(* IEC 61131-3 sources: Industry-PLC-LLM/data/PLCBEAD_repo/PLCBEAD_PLCEmbed-main/PLC-BEAD/Source/OpenPLCv2 (part 8) *)

(* ---- REPLACE_CHARS.ST ---- *)
FUNCTION_BLOCK REPLACE_CHARS_Block

	VAR_INPUT
		STR :	STRING;
		SRC :	STRING;
		REP :	STRING;
	END_VAR

	VAR_OUTPUT
		REPLACE_CHARS :	STRING;
	END_VAR

	VAR
		tmp :	STRING;
		a :	INT;
		b :	INT;
		c :	STRING;
		stp :	INT;
	END_VAR

	REPLACE_CHARS := STR;

	a := LEN(src);
	b := LEN(rep);
	IF a < b THEN
		rep := LEFT(rep, a);
	ELSIF b < a THEN
		src := LEFT(src, b);
	END_IF;

	stp := LEN(str);
	FOR a := 1 TO stp DO
		c := MID(REPLACE_CHARS, 1, a);
		b := FIND(src, c);
		IF b > 0 THEN
			tmp := MID(rep, 1, b);
			REPLACE_CHARS := REPLACE(REPLACE_CHARS, tmp, 1, a);
		END_IF;
	END_FOR;

END_FUNCTION_BLOCK

PROGRAM program0

	VAR
		STR :	STRING;
		SRC :	STRING;
		REP :	STRING;

        REPLACE_CHARS :	STRING;
		func_block : REPLACE_CHARS_Block;
	END_VAR
		func_block.STR := STR;
		func_block.SRC := SRC;
		func_block.REP := REP;
		func_block();
		REPLACE_CHARS := func_block.REPLACE_CHARS;

END_PROGRAM

CONFIGURATION Config0

	RESOURCE Res0 ON PLC
		TASK task0(INTERVAL := T#20ms,PRIORITY := 0);
		PROGRAM instance0 WITH task0 : program0;
	END_RESOURCE

END_CONFIGURATION

(* ---- RMP_B.ST ---- *)
FUNCTION TIME_TO_UDINT2:UDINT
	VAR_INPUT
		X :	TIME;
	END_VAR

	TIME_TO_UDINT2 := DINT_TO_UDINT(TIME_TO_DINT(X));
END_FUNCTION

FUNCTION_BLOCK T_PLC_MS_block
	VAR_OUTPUT
		T_PLC_MS :	UDINT;
	END_VAR

	VAR_EXTERNAL
		PLC_TICKS_PER_SEC :	INT;
		PLC_SYS_TICK_CNT :	DINT;
	END_VAR

	VAR
		debug :	BOOL;(*Debug-Mode ON / OFF*)
		N :	INT;(*Debug-Faktor*)
		Offset :	UDINT;(*Debug-Offset*)
		temp :	DWORD := DWORD#1;(*Debug-Offset*)
		mode :	BOOL;(*modus*)
		faktor :	UDINT;(*Systemtakt-Faktor*)
		init :	BOOL;
		v_plc_ticks_per_sec :	UDINT;
		base :	UDINT := UDINT#1000;
	END_VAR

	IF init = FALSE THEN
		v_plc_ticks_per_sec := INT_TO_UDINT(PLC_TICKS_PER_SEC);
		IF v_plc_ticks_per_sec = UDINT#1024 THEN
			faktor := UDINT#1;
			mode := FALSE;
		ELSIF v_plc_ticks_per_sec > UDINT#0 THEN
			IF v_plc_ticks_per_sec <= base THEN
				faktor := base / v_plc_ticks_per_sec;
				mode := FALSE;
			ELSE
				faktor := v_plc_ticks_per_sec / base;
				mode := TRUE;
			END_IF;
		ELSE
			faktor := UDINT#1;
		END_IF;
		init := TRUE;
	END_IF;

	IF mode THEN
		T_PLC_MS := DINT_TO_UDINT(PLC_SYS_TICK_CNT) / faktor;
	ELSE
		T_PLC_MS := DINT_TO_UDINT(PLC_SYS_TICK_CNT) * faktor;
	END_IF;

	IF debug THEN
		T_PLC_MS := (DWORD_TO_UDINT(SHL(UDINT_TO_DWORD(T_PLC_MS),N) OR SHL(temp,N)) - UDINT#1) + Offset;
	END_IF;
END_FUNCTION_BLOCK

FUNCTION FRMP_B:BYTE
	VAR_INPUT
		START :	BYTE;
		DIR :	BOOL;
		TD :	TIME;
		TR :	TIME;
	END_VAR

	IF TD < TR THEN
		FRMP_B := MIN(UDINT_TO_BYTE(DWORD_TO_UDINT(SHL(TIME_TO_DWORD(TD), 8)) / TIME_TO_UDINT2(TR)), SEL(DIR, START, USINT_TO_BYTE(USINT#255 - BYTE_TO_USINT(START))));
		IF DIR THEN
			FRMP_B := USINT_TO_BYTE(BYTE_TO_USINT(START) + BYTE_TO_USINT(FRMP_B));
		ELSE
			FRMP_B := USINT_TO_BYTE(BYTE_TO_USINT(START) - BYTE_TO_USINT(FRMP_B));
		END_IF;
	ELSE
		FRMP_B := SEL(DIR, BYTE#0, BYTE#255);
	END_IF;
END_FUNCTION

FUNCTION_BLOCK _RMP_B
	VAR_INPUT
		DIR :	BOOL;
		E :	BOOL := TRUE;
		TR :	TIME;
	END_VAR

	VAR_IN_OUT
		RMP :	BYTE;
	END_VAR

	VAR
		T_PLC_MS :	T_PLC_MS_block;
		tx :	TIME;
		tl :	TIME;
		tn :	TIME;
		init :	BOOL;
		last_dir :	BOOL;
		start :	BYTE;
	END_VAR

	T_PLC_MS();
	tx := UDINT_TO_TIME(T_PLC_MS.T_PLC_MS);

	IF E AND init AND (dir = last_dir) AND (RMP <> SEL(DIR, BYTE#0, BYTE#255)) AND TR = tn THEN
		RMP := FRMP_B(start, DIR, tx - tl, TR);
	ELSE
		init := TRUE;
		tl := tx;
		tn := tr;
		start := RMP;
	END_IF;
	last_dir := dir;
END_FUNCTION_BLOCK

FUNCTION_BLOCK RMP_B_Block

	VAR_INPUT
		SET :	BOOL;
		PT :	TIME;
		E :	BOOL := TRUE;
		UP :	BOOL := TRUE;
		RST :	BOOL;
	END_VAR

	VAR_OUTPUT
		OUT :	BYTE;
		BUSY :	BOOL;
		HIGH :	BOOL;
		LOW :	BOOL;
	END_VAR

	VAR
		rmp :	_RMP_B;
	END_VAR

	rmp(dir := UP, E := E, TR := PT, RMP := out);
	out := rmp.RMP;

	IF RST THEN
		out := BYTE#0;
	ELSIF SET THEN
		out := BYTE#255;
	END_IF;

low := out = BYTE#0;
high := out = BYTE#255;
busy := NOT (low OR high) AND E;

END_FUNCTION_BLOCK

PROGRAM program0
	VAR
		SET :	BOOL;
		PT :	TIME;
		E :	BOOL := TRUE;
		UP :	BOOL := TRUE;
		RST :	BOOL;

		OUT :	BYTE;
		BUSY :	BOOL;
		HIGH :	BOOL;
		LOW :	BOOL;

		func_block : RMP_B_Block;
	END_VAR
		func_block.SET := SET;
		func_block.PT := PT;
		func_block.E := E;
		func_block.UP := UP;
		func_block.RST := RST;
		func_block();
		OUT := func_block.OUT;
		BUSY := func_block.BUSY;
		HIGH := func_block.HIGH;
		LOW := func_block.LOW;

END_PROGRAM

CONFIGURATION Config0
	VAR_GLOBAL
		PLC_TICKS_PER_SEC :	INT;
		PLC_SYS_TICK_CNT :	DINT;
	END_VAR

  	RESOURCE Res0 ON PLC
    	TASK task0(INTERVAL := T#20ms,PRIORITY := 0);
    	PROGRAM instance0 WITH task0 : program0;
  	END_RESOURCE
END_CONFIGURATION

(* ---- RMP_SOFT.ST ---- *)
FUNCTION TIME_TO_UDINT2:UDINT
	VAR_INPUT
		X :	TIME;
	END_VAR

	TIME_TO_UDINT2 := DINT_TO_UDINT(TIME_TO_DINT(X));
END_FUNCTION

FUNCTION_BLOCK T_PLC_MS_block
	VAR_OUTPUT
		T_PLC_MS :	UDINT;
	END_VAR

	VAR_EXTERNAL
		PLC_TICKS_PER_SEC :	INT;
		PLC_SYS_TICK_CNT :	DINT;
	END_VAR

	VAR
		debug :	BOOL;(*Debug-Mode ON / OFF*)
		N :	INT;(*Debug-Faktor*)
		Offset :	UDINT;(*Debug-Offset*)
		temp :	DWORD := DWORD#1;(*Debug-Offset*)
		mode :	BOOL;(*modus*)
		faktor :	UDINT;(*Systemtakt-Faktor*)
		init :	BOOL;
		v_plc_ticks_per_sec :	UDINT;
		base :	UDINT := UDINT#1000;
	END_VAR

	IF init = FALSE THEN
		v_plc_ticks_per_sec := INT_TO_UDINT(PLC_TICKS_PER_SEC);
		IF v_plc_ticks_per_sec = UDINT#1024 THEN
			faktor := UDINT#1;
			mode := FALSE;
		ELSIF v_plc_ticks_per_sec > UDINT#0 THEN
			IF v_plc_ticks_per_sec <= base THEN
				faktor := base / v_plc_ticks_per_sec;
				mode := FALSE;
			ELSE
				faktor := v_plc_ticks_per_sec / base;
				mode := TRUE;
			END_IF;
		ELSE
			faktor := UDINT#1;
		END_IF;
		init := TRUE;
	END_IF;

	IF mode THEN
		T_PLC_MS := DINT_TO_UDINT(PLC_SYS_TICK_CNT) / faktor;
	ELSE
		T_PLC_MS := DINT_TO_UDINT(PLC_SYS_TICK_CNT) * faktor;
	END_IF;

	IF debug THEN
		T_PLC_MS := (DWORD_TO_UDINT(SHL(UDINT_TO_DWORD(T_PLC_MS),N) OR SHL(temp,N)) - UDINT#1) + Offset;
	END_IF;
END_FUNCTION_BLOCK

FUNCTION FRMP_B:BYTE
	VAR_INPUT
		START :	BYTE;
		DIR :	BOOL;
		TD :	TIME;
		TR :	TIME;
	END_VAR

	IF TD < TR THEN
		FRMP_B := MIN(UDINT_TO_BYTE(DWORD_TO_UDINT(SHL(TIME_TO_DWORD(TD), 8)) / TIME_TO_UDINT2(TR)), SEL(DIR, START, USINT_TO_BYTE(USINT#255 - BYTE_TO_USINT(START))));
		IF DIR THEN
			FRMP_B := USINT_TO_BYTE(BYTE_TO_USINT(START) + BYTE_TO_USINT(FRMP_B));
		ELSE
			FRMP_B := USINT_TO_BYTE(BYTE_TO_USINT(START) - BYTE_TO_USINT(FRMP_B));
		END_IF;
	ELSE
		FRMP_B := SEL(DIR, BYTE#0, BYTE#255);
	END_IF;
END_FUNCTION

FUNCTION_BLOCK _RMP_B
	VAR_INPUT
		DIR :	BOOL;
		E :	BOOL := TRUE;
		TR :	TIME;
	END_VAR

	VAR_IN_OUT
		RMP :	BYTE;
	END_VAR

	VAR
		T_PLC_MS :	T_PLC_MS_block;
		tx :	TIME;
		tl :	TIME;
		tn :	TIME;
		init :	BOOL;
		last_dir :	BOOL;
		start :	BYTE;
	END_VAR

	T_PLC_MS();
	tx := UDINT_TO_TIME(T_PLC_MS.T_PLC_MS);

	IF E AND init AND (dir = last_dir) AND (RMP <> SEL(DIR, BYTE#0, BYTE#255)) AND TR = tn THEN
		RMP := FRMP_B(start, DIR, tx - tl, TR);
	ELSE
		init := TRUE;
		tl := tx;
		tn := tr;
		start := RMP;
	END_IF;
	last_dir := dir;
END_FUNCTION_BLOCK

FUNCTION_BLOCK RMP_SOFT_Block

	VAR_INPUT
		IN :	BOOL;
		VAL :	BYTE;
		PT_ON :	TIME := T#100ms;
		PT_OFF :	TIME := T#100ms;
	END_VAR

	VAR_OUTPUT
		OUT :	BYTE := BYTE#00;
	END_VAR

	VAR
		rmp :	_RMP_B;
		tmp :	BYTE;
	END_VAR

	tmp := SEL(in, BYTE#0, val);
	IF tmp > out THEN
		(* we need to ramp down *)
		rmp(dir := TRUE, E := TRUE, TR := PT_ON, RMP := out);
		out := rmp.RMP;
		(* make sure out does not surpass tmp *)
		out := MIN(out, tmp);
	ELSIF tmp < out THEN
		(* we need to ramp up *)
		rmp(dir := FALSE, E := TRUE, TR := PT_OFF, RMP := out);
		out := rmp.RMP;
		(* make sure out does not surpass tmp *)
		out := MAX(out, tmp);
	ELSE
		(* no ramp necessary *)
		rmp(E := FALSE, RMP := out);
		out := rmp.RMP;
	END_IF;

END_FUNCTION_BLOCK

PROGRAM program0
	VAR
		IN :	BOOL;
		VAL :	BYTE;
		PT_ON :	TIME;
		PT_OFF : TIME;

		OUT  :	BYTE;

		func_block : RMP_SOFT_Block;
	END_VAR
		func_block.IN := IN;
		func_block.VAL := VAL;
		func_block.PT_ON := PT_ON;
		func_block.PT_OFF := PT_OFF;
		func_block();
		OUT  := func_block.OUT ;

END_PROGRAM

CONFIGURATION Config0
	VAR_GLOBAL
		PLC_TICKS_PER_SEC :	INT;
		PLC_SYS_TICK_CNT :	DINT;
	END_VAR

  	RESOURCE Res0 ON PLC
    	TASK task0(INTERVAL := T#20ms,PRIORITY := 0);
    	PROGRAM instance0 WITH task0 : program0;
  	END_RESOURCE
END_CONFIGURATION

(* ---- RMP_W.ST ---- *)
FUNCTION_BLOCK T_PLC_MS_block
	VAR_OUTPUT
		T_PLC_MS :	UDINT;
	END_VAR

	VAR_EXTERNAL
		PLC_TICKS_PER_SEC :	INT;
		PLC_SYS_TICK_CNT :	DINT;
	END_VAR

	VAR
		debug :	BOOL;(*Debug-Mode ON / OFF*)
		N :	INT;(*Debug-Faktor*)
		Offset :	UDINT;(*Debug-Offset*)
		temp :	DWORD := DWORD#1;(*Debug-Offset*)
		mode :	BOOL;(*modus*)
		faktor :	UDINT;(*Systemtakt-Faktor*)
		init :	BOOL;
		v_plc_ticks_per_sec :	UDINT;
		base :	UDINT := UDINT#1000;
	END_VAR

	IF init = FALSE THEN
		v_plc_ticks_per_sec := INT_TO_UDINT(PLC_TICKS_PER_SEC);
		IF v_plc_ticks_per_sec = UDINT#1024 THEN
			faktor := UDINT#1;
			mode := FALSE;
		ELSIF v_plc_ticks_per_sec > UDINT#0 THEN
			IF v_plc_ticks_per_sec <= base THEN
				faktor := base / v_plc_ticks_per_sec;
				mode := FALSE;
			ELSE
				faktor := v_plc_ticks_per_sec / base;
				mode := TRUE;
			END_IF;
		ELSE
			faktor := UDINT#1;
		END_IF;
		init := TRUE;
	END_IF;

	IF mode THEN
		T_PLC_MS := DINT_TO_UDINT(PLC_SYS_TICK_CNT) / faktor;
	ELSE
		T_PLC_MS := DINT_TO_UDINT(PLC_SYS_TICK_CNT) * faktor;
	END_IF;

	IF debug THEN
		T_PLC_MS := (DWORD_TO_UDINT(SHL(UDINT_TO_DWORD(T_PLC_MS),N) OR SHL(temp,N)) - UDINT#1) + Offset;
	END_IF;
END_FUNCTION_BLOCK

FUNCTION _WORD_TO_DINT:DINT
	VAR_INPUT
		IN :	WORD;
	END_VAR
	_WORD_TO_DINT := UINT_TO_DINT(WORD_TO_UINT(IN));
END_FUNCTION

FUNCTION TIME_TO_UDINT2:UDINT
	VAR_INPUT
		X :	TIME;
	END_VAR

	TIME_TO_UDINT2 := DINT_TO_UDINT(TIME_TO_DINT(X));
END_FUNCTION

FUNCTION_BLOCK _RMP_W

	VAR_INPUT
		DIR :	BOOL;
		E :	BOOL := TRUE;
		TR :	TIME;
	END_VAR

	VAR_IN_OUT
		RMP :	WORD;
	END_VAR

	VAR
		T_PLC_MS :	T_PLC_MS_block;
		tx :	UDINT;
		tl :	UDINT;
		ptesss :	DINT;
		init :	BOOL;
		last_dir :	BOOL;
	END_VAR

	T_PLC_MS();
	tx := T_PLC_MS.T_PLC_MS;
	IF E AND init THEN
		(* we need to set tl = tx when direction changes *)
		IF dir XOR last_dir THEN
			tl := tx;
			last_dir := dir;
		END_IF;
		(* check_elapsed time and calculate only if necessary *)
		IF tr > t#0s THEN
			ptesss := DWORD_TO_DINT(UDINT_TO_DWORD(DWORD_TO_UDINT(SHL(UDINT_TO_DWORD(tx-tl), 16)) / TIME_TO_UDINT2(TR)));
		ELSE
			ptesss := DINT#65535;
		END_IF;
		IF ptesss > DINT#0 THEN
			(* perform the ptesss on the ramp *)
			tl := tx;
			(* calculate the ptesss response *)
			IF NOT dir THEN ptesss := - ptesss; END_IF;
			rmp := DINT_TO_WORD(LIMIT(DINT#0, _WORD_TO_DINT(rmp) + ptesss, DINT#65535));
		END_IF;
	ELSE
		tl := tx;
		init := TRUE;
	END_IF;
END_FUNCTION_BLOCK

FUNCTION_BLOCK RMP_W

	VAR_INPUT
		SET :	BOOL;
		PT :	TIME;
		E :	BOOL := TRUE;
		UP :	BOOL := TRUE;
		RST :	BOOL;
	END_VAR

	VAR_OUTPUT
		OUT :	WORD;
		BUSY :	BOOL;
		HIGH :	BOOL;
		LOW :	BOOL;
	END_VAR

	VAR
		rmp :	_RMP_W;
	END_VAR

	rmp(dir := UP, E := E, TR := PT, rmp := out);
	out := rmp.RMP;

	IF RST THEN
		out := WORD#0;
	ELSIF SET THEN
		out := WORD#65535;
	END_IF;

	low := out = WORD#0;
	high := out = WORD#65535;
	busy := NOT (low OR high) AND E;

END_FUNCTION_BLOCK

PROGRAM program0
  VAR
		SET :	BOOL;
		PT  :	TIME;
		E   :	BOOL;
		UP  :	BOOL ;
		RST :	BOOL;

		OUT  :	WORD;
		BUSY :	BOOL;
		HIGH :	BOOL;
		LOW  :	BOOL;

	func_block : RMP_W;
  END_VAR
	func_block.SET:=SET;
	func_block.PT :=PT ;
	func_block.E  :=E ;
	func_block.UP :=UP ;
	func_block.RST:=RST;
	func_block();
	OUT  := func_block.OUT ;
	BUSY := func_block.BUSY;
	HIGH := func_block.HIGH;
	LOW  := func_block.LOW ;

END_PROGRAM

CONFIGURATION Config0
	VAR_GLOBAL
		PLC_TICKS_PER_SEC :	INT;
		PLC_SYS_TICK_CNT :	DINT;
	END_VAR
  	RESOURCE Res0 ON PLC
    	TASK task0(INTERVAL := T#20ms,PRIORITY := 0);
    	PROGRAM instance0 WITH task0 : program0;
  	END_RESOURCE
END_CONFIGURATION

(* ---- RTC_2.ST ---- *)
FUNCTION _INT_TO_UDINT:UDINT
	VAR_INPUT
		IN :	INT;
	END_VAR

	_INT_TO_UDINT := DINT_TO_UDINT(INT_TO_DINT(IN));
END_FUNCTION

FUNCTION SET_DATE:UDINT

	VAR_INPUT
		YEAR :	INT;
		MONTH :	INT;
		DAY :	INT;
	END_VAR

	VAR
		count :	INT;
	END_VAR

	IF month > 2 THEN
		count := (month - 1) * 30;
		IF month > 7 THEN
			count := count + DWORD_TO_INT(SHR(DINT_TO_DWORD(INT_TO_DINT(month) - INT_TO_DINT(3)),1));
		ELSE
			count := count + DWORD_TO_INT(SHR(DINT_TO_DWORD(INT_TO_DINT(month) - INT_TO_DINT(4)),1));
		END_IF;
		IF SHL(INT_TO_WORD(year),14) = WORD#0 THEN
			count := count + 1;
		END_IF;
	ELSE
		count := (month - 1) * 31;
	END_IF;
	SET_DATE := (_INT_TO_UDINT(count + day - 1) + DWORD_TO_UDINT(SHR(UDINT_TO_DWORD(_INT_TO_UDINT(year) * UDINT#1461 - UDINT#2878169), 2))) * UDINT#86400;

END_FUNCTION

FUNCTION SET_DT:UDINT
	VAR_INPUT
		YEAR :	INT;
		MONTH :	INT;
		DAY :	INT;
		HOUR :	INT;
		MINUTE :	INT;
		SECOND :	INT;
	END_VAR

	SET_DT := SET_DATE(YEAR, MONTH, DAY) + _INT_TO_UDINT(SECOND) + _INT_TO_UDINT(MINUTE) * UDINT#60 + _INT_TO_UDINT(HOUR) * UDINT#3600;
END_FUNCTION

FUNCTION DT_TO_DATE2:UDINT

	VAR_INPUT
		IN :	UDINT;
	END_VAR

	DT_TO_DATE2 := (IN / UDINT#86400) * UDINT#86400;

END_FUNCTION

FUNCTION YEAR_OF_DATE:INT
	VAR_INPUT
		IDATE :	UDINT;
	END_VAR

	YEAR_OF_DATE := UDINT_TO_INT((idate+UDINT#43200) / UDINT#31557600 + UDINT#1970);
END_FUNCTION

FUNCTION DST:BOOL
	VAR_INPUT
		UTC :	UDINT;
	END_VAR

	VAR
		yr :	INT;
		yr4 :	UDINT;
		ltc :	UDINT;
		idate :	UDINT;
	END_VAR

	yr := YEAR_OF_DATE(DT_TO_DATE2(UTC));
	ltc := UTC;
	idate := SET_DT(yr, 3, 31, 1, 0, 0);
	yr4 := DWORD_TO_UDINT(SHR(INT_TO_DWORD(5 * yr), 2)) + UDINT#1;
	DST := (idate - ((yr4 + UDINT#3) MOD UDINT#7) * UDINT#86400 <= ltc) AND (idate + (UDINT#214 - (yr4) MOD UDINT#7) * UDINT#86400 > ltc);

END_FUNCTION

FUNCTION_BLOCK T_PLC_MS_Block
	VAR_OUTPUT
		T_PLC_MS :	UDINT;
	END_VAR

	VAR_EXTERNAL
		PLC_TICKS_PER_SEC :	INT;
		PLC_SYS_TICK_CNT :	DINT;
	END_VAR

	VAR
		debug :	BOOL;(*Debug-Mode ON / OFF*)
		N :	INT;(*Debug-Faktor*)
		Offset :	UDINT;(*Debug-Offset*)
		temp :	DWORD := DWORD#1;(*Debug-Offset*)
		mode :	BOOL;(*modus*)
		faktor :	UDINT;(*Systemtakt-Faktor*)
		init :	BOOL;
		v_plc_ticks_per_sec :	UDINT;
		base :	UDINT := UDINT#1000;
	END_VAR

	IF init = FALSE THEN
		v_plc_ticks_per_sec := INT_TO_UDINT(PLC_TICKS_PER_SEC);
		IF v_plc_ticks_per_sec = UDINT#1024 THEN
			faktor := UDINT#1;
			mode := FALSE;
		ELSIF v_plc_ticks_per_sec > UDINT#0 THEN
			IF v_plc_ticks_per_sec <= base THEN
				faktor := base / v_plc_ticks_per_sec;
				mode := FALSE;
			ELSE
				faktor := v_plc_ticks_per_sec / base;
				mode := TRUE;
			END_IF;
		ELSE
			faktor := UDINT#1;
		END_IF;
		init := TRUE;
	END_IF;

	IF mode THEN
		T_PLC_MS := DINT_TO_UDINT(PLC_SYS_TICK_CNT) / faktor;
	ELSE
		T_PLC_MS := DINT_TO_UDINT(PLC_SYS_TICK_CNT) * faktor;
	END_IF;

	IF debug THEN
		T_PLC_MS := (DWORD_TO_UDINT(SHL(UDINT_TO_DWORD(T_PLC_MS),N) OR SHL(temp,N)) - UDINT#1) + Offset;
	END_IF;
END_FUNCTION_BLOCK

FUNCTION_BLOCK RTC_MS_Block

	VAR_INPUT
		SET :	BOOL;
		SDT :	UDINT;
		SMS :	INT;
	END_VAR

	VAR_OUTPUT
		XDT :	UDINT;
		XMS :	INT;
	END_VAR

	VAR
		init :	BOOL;
		last :	UDINT;
		tx :	UDINT;
		T_PLC_MS :	T_PLC_MS_Block;
	END_VAR

	T_PLC_MS();
	tx:= T_PLC_MS.T_PLC_MS;

	IF set OR NOT init THEN
		(* clock needs to be set when set is true or after power up *)
		init := TRUE;
		xdt := SDT;
		XMS := SMS;
	ELSE
		XMS := XMS + UDINT_TO_INT(tx - last);
		(* check if one second has expired *)
		IF XMS > 999 THEN
			XDT := XDT + UDINT#1; (* add one second *)
			XMS := XMS - 1000;
		END_IF;
	END_IF;
	last := tx;

END_FUNCTION_BLOCK

FUNCTION_BLOCK RTC_2_Block

	VAR_INPUT
		SET :	BOOL;
		SDT :	UDINT;
		SMS :	INT;
		DEN :	BOOL;
		OFS :	INT;
	END_VAR

	VAR_OUTPUT
		UDT :	UDINT;
		LDT :	UDINT;
		DSO :	BOOL;
		XMS :	INT;
	END_VAR

	VAR
		RT :	RTC_MS_Block;
	END_VAR

	RT(SET := SET, SDT := SDT, SMS := SMS);
	UDT := rt.xdt;
	XMS := rt.XMS;

	dso := DST(udt) AND DEN;

	LDT := UDT + _INT_TO_UDINT(ofs + BOOL_TO_INT(DSO) * 60) * UDINT#60;

END_FUNCTION_BLOCK

PROGRAM program0

	VAR
		SET :	BOOL;
		SDT :	UDINT;
		SMS :	INT;
		DEN :	BOOL;
		OFS :	INT;
		UDT :	UDINT;
		LDT :	UDINT;
		DSO :	BOOL;
		XMS :	INT;
		func_block : RTC_2_Block;
  	END_VAR
	func_block.SET  :=	SET;
	func_block.SDT  :=	SDT;
	func_block.SMS  :=	SMS;
	func_block.DEN  :=	DEN;
	func_block.OFS  :=	OFS;
	func_block();
	UDT := func_block.UDT;
	LDT := func_block.LDT;
	DSO := func_block.DSO;
	XMS := func_block.XMS;

END_PROGRAM

CONFIGURATION Config0

	VAR_GLOBAL
		PLC_TICKS_PER_SEC :	INT;
		PLC_SYS_TICK_CNT :	DINT;
	END_VAR

	RESOURCE Res0 ON PLC
		TASK task0(INTERVAL := T#20ms,PRIORITY := 0);
		PROGRAM instance0 WITH task0 : program0;
	END_RESOURCE

END_CONFIGURATION

(* ---- RTC_MS.ST ---- *)
FUNCTION_BLOCK T_PLC_MS_Block
	VAR_OUTPUT
		T_PLC_MS :	UDINT;
	END_VAR

	VAR_EXTERNAL
		PLC_TICKS_PER_SEC :	INT;
		PLC_SYS_TICK_CNT :	DINT;
	END_VAR

	VAR
		debug :	BOOL;(*Debug-Mode ON / OFF*)
		N :	INT;(*Debug-Faktor*)
		Offset :	UDINT;(*Debug-Offset*)
		temp :	DWORD := DWORD#1;(*Debug-Offset*)
		mode :	BOOL;(*modus*)
		faktor :	UDINT;(*Systemtakt-Faktor*)
		init :	BOOL;
		v_plc_ticks_per_sec :	UDINT;
		base :	UDINT := UDINT#1000;
	END_VAR

	IF init = FALSE THEN
		v_plc_ticks_per_sec := INT_TO_UDINT(PLC_TICKS_PER_SEC);
		IF v_plc_ticks_per_sec = UDINT#1024 THEN
			faktor := UDINT#1;
			mode := FALSE;
		ELSIF v_plc_ticks_per_sec > UDINT#0 THEN
			IF v_plc_ticks_per_sec <= base THEN
				faktor := base / v_plc_ticks_per_sec;
				mode := FALSE;
			ELSE
				faktor := v_plc_ticks_per_sec / base;
				mode := TRUE;
			END_IF;
		ELSE
			faktor := UDINT#1;
		END_IF;
		init := TRUE;
	END_IF;

	IF mode THEN
		T_PLC_MS := DINT_TO_UDINT(PLC_SYS_TICK_CNT) / faktor;
	ELSE
		T_PLC_MS := DINT_TO_UDINT(PLC_SYS_TICK_CNT) * faktor;
	END_IF;

	IF debug THEN
		T_PLC_MS := (DWORD_TO_UDINT(SHL(UDINT_TO_DWORD(T_PLC_MS),N) OR SHL(temp,N)) - UDINT#1) + Offset;
	END_IF;
END_FUNCTION_BLOCK

FUNCTION_BLOCK RTC_MS_Block

	VAR_INPUT
		SET :	BOOL;
		SDT :	UDINT;
		SMS :	INT;
	END_VAR

	VAR_OUTPUT
		XDT :	UDINT;
		XMS :	INT;
	END_VAR

	VAR
		init :	BOOL;
		last :	UDINT;
		tx :	UDINT;
		T_PLC_MS :	T_PLC_MS_Block;
	END_VAR

	T_PLC_MS();
	tx:= T_PLC_MS.T_PLC_MS;

	IF set OR NOT init THEN
		(* clock needs to be set when set is true or after power up *)
		init := TRUE;
		xdt := SDT;
		XMS := SMS;
	ELSE
		XMS := XMS + UDINT_TO_INT(tx - last);
		(* check if one second has expired *)
		IF XMS > 999 THEN
			XDT := XDT + UDINT#1; (* add one second *)
			XMS := XMS - 1000;
		END_IF;
	END_IF;
	last := tx;

END_FUNCTION_BLOCK

PROGRAM program0

	VAR
		SET :	BOOL;
		SDT :	UDINT;
		SMS :	INT;
		XDT :	UDINT;
		XMS :	INT;
		func_block : RTC_MS_Block;
  	END_VAR
	func_block.SET  :=	SET;
	func_block.SDT  :=	SDT;
	func_block.SMS  :=	SMS;
	func_block();
	XDT := func_block.XDT;
	XMS := func_block.XMS;

END_PROGRAM

CONFIGURATION Config0

	VAR_GLOBAL
		PLC_TICKS_PER_SEC :	INT;
		PLC_SYS_TICK_CNT :	DINT;
	END_VAR

	RESOURCE Res0 ON PLC
		TASK task0(INTERVAL := T#20ms,PRIORITY := 0);
		PROGRAM instance0 WITH task0 : program0;
	END_RESOURCE

END_CONFIGURATION

(* ---- SCHEDULER.ST ---- *)
FUNCTION_BLOCK T_PLC_MS_block
	VAR_OUTPUT
		T_PLC_MS :	UDINT;
	END_VAR

	VAR_EXTERNAL
		PLC_TICKS_PER_SEC :	INT;
		PLC_SYS_TICK_CNT :	DINT;
	END_VAR

	VAR
		debug :	BOOL;(*Debug-Mode ON / OFF*)
		N :	INT;(*Debug-Faktor*)
		Offset :	UDINT;(*Debug-Offset*)
		temp :	DWORD := DWORD#1;(*Debug-Offset*)
		mode :	BOOL;(*modus*)
		faktor :	UDINT;(*Systemtakt-Faktor*)
		init :	BOOL;
		v_plc_ticks_per_sec :	UDINT;
		base :	UDINT := UDINT#1000;
	END_VAR

	IF init = FALSE THEN
		v_plc_ticks_per_sec := INT_TO_UDINT(PLC_TICKS_PER_SEC);
		IF v_plc_ticks_per_sec = UDINT#1024 THEN
			faktor := UDINT#1;
			mode := FALSE;
		ELSIF v_plc_ticks_per_sec > UDINT#0 THEN
			IF v_plc_ticks_per_sec <= base THEN
				faktor := base / v_plc_ticks_per_sec;
				mode := FALSE;
			ELSE
				faktor := v_plc_ticks_per_sec / base;
				mode := TRUE;
			END_IF;
		ELSE
			faktor := UDINT#1;
		END_IF;
		init := TRUE;
	END_IF;

	IF mode THEN
		T_PLC_MS := DINT_TO_UDINT(PLC_SYS_TICK_CNT) / faktor;
	ELSE
		T_PLC_MS := DINT_TO_UDINT(PLC_SYS_TICK_CNT) * faktor;
	END_IF;

	IF debug THEN
		T_PLC_MS := (DWORD_TO_UDINT(SHL(UDINT_TO_DWORD(T_PLC_MS),N) OR SHL(temp,N)) - UDINT#1) + Offset;
	END_IF;
END_FUNCTION_BLOCK

FUNCTION_BLOCK SCHEDULER_Block

	VAR_INPUT
		E0 :	BOOL;
		E1 :	BOOL;
		E2 :	BOOL;
		E3 :	BOOL;
		T0 :	TIME;
		T1 :	TIME;
		T2 :	TIME;
		T3 :	TIME;
	END_VAR

	VAR_OUTPUT
		Q0 :	BOOL;
		Q1 :	BOOL;
		Q2 :	BOOL;
		Q3 :	BOOL;
	END_VAR

	VAR
		T_PLC_MS :	T_PLC_MS_Block;
		init :	BOOL;
		s0 :	TIME;
		s1 :	TIME;
		s2 :	TIME;
		s3 :	TIME;
		tx :	TIME;
		c :	INT;
	END_VAR

	T_PLC_MS();
	tx:= UDINT_TO_TIME(T_PLC_MS.T_PLC_MS);

	IF NOT init THEN
		init := TRUE;
		s0 := tx - T0;
		s1 := tx - T1;
		s2 := tx - T2;
		s3 := tx - T3;
	END_IF;

	Q0 := FALSE;
	Q1 := FALSE;
	Q2 := FALSE;
	Q3 := FALSE;

	CASE c OF
		0: 	IF tx - s0 >= T0 THEN
				Q0 := E0;
				s0 := tx;
			END_IF;
			c := 1;
		1: 	IF tx - s1 >= T1 THEN
				Q1 := E1;
				s1 := tx;
			END_IF;
			c := 2;
		2: 	IF tx - s2 >= T2 THEN
				Q2 := E2;
				s2 := tx;
			END_IF;
			c := 3;
		3: 	IF tx - s3 >= T3 THEN
				Q3 := E3;
				s3 := tx;
			END_IF;
			c := 0;
	END_CASE;

END_FUNCTION_BLOCK

PROGRAM program0

	VAR
		E0 :	BOOL;
		E1 :	BOOL;
		E2 :	BOOL;
		E3 :	BOOL;
		T0 :	TIME;
		T1 :	TIME;
		T2 :	TIME;
		T3 :	TIME;
		Q0 :	BOOL;
		Q1 :	BOOL;
		Q2 :	BOOL;
		Q3 :	BOOL;
		func_block : SCHEDULER_Block;
  	END_VAR
	func_block.E0  :=	E0;
	func_block.E1  :=	E1;
	func_block.E2  :=	E2;
	func_block.E3  :=	E3;
	func_block.T0  :=	T0;
	func_block.T1  :=	T1;
	func_block.T2  :=	T2;
	func_block.T3  :=	T3;
	func_block();
	Q0 := func_block.Q0;
	Q1 := func_block.Q1;
	Q2 := func_block.Q2;
	Q3 := func_block.Q3;

END_PROGRAM

CONFIGURATION Config0
	VAR_GLOBAL
		PLC_TICKS_PER_SEC :	INT;
		PLC_SYS_TICK_CNT :	DINT;
	END_VAR
	RESOURCE Res0 ON PLC
		TASK task0(INTERVAL := T#20ms,PRIORITY := 0);
		PROGRAM instance0 WITH task0 : program0;
	END_RESOURCE
END_CONFIGURATION

(* ---- SCHEDULER_2.ST ---- *)
FUNCTION_BLOCK SCHEDULER_2_Block

	VAR_INPUT
		E0 :	BOOL;
		E1 :	BOOL;
		E2 :	BOOL;
		E3 :	BOOL;
		C0 :	UINT;
		C1 :	UINT;
		C2 :	UINT;
		C3 :	UINT;
		O0 :	UINT;
		O1 :	UINT;
		O2 :	UINT;
		O3 :	UINT;
	END_VAR

	VAR_OUTPUT
		Q0 :	BOOL;
		Q1 :	BOOL;
		Q2 :	BOOL;
		Q3 :	BOOL;
	END_VAR

	VAR
		sx :	UINT;
	END_VAR

	Q0 := E0 AND (sx MOD C0 - O0 = UINT#0);
	Q1 := E1 AND (sx MOD C1 - O1 = UINT#0);
	Q2 := E2 AND (sx MOD C2 - O2 = UINT#0);
	Q3 := E3 AND (sx MOD C3 - O3 = UINT#0);

	sx := sx + UINT#1;

END_FUNCTION_BLOCK

PROGRAM program0

	VAR
		E0 :	BOOL;
		E1 :	BOOL;
		E2 :	BOOL;
		E3 :	BOOL;
		C0 :	UINT;
		C1 :	UINT;
		C2 :	UINT;
		C3 :	UINT;
		O0 :	UINT;
		O1 :	UINT;
		O2 :	UINT;
		O3 :	UINT;
		Q0 :	BOOL;
		Q1 :	BOOL;
		Q2 :	BOOL;
		Q3 :	BOOL;
		func_block : SCHEDULER_2_Block;
  	END_VAR
	func_block.E0  :=	E0;
	func_block.E1  :=	E1;
	func_block.E2  :=	E2;
	func_block.E3  :=	E3;
	func_block.C0  :=	C0;
	func_block.C1  :=	C1;
	func_block.C2  :=	C2;
	func_block.C3  :=	C3;
	func_block.O0  :=	O0;
	func_block.O1  :=	O1;
	func_block.O2  :=	O2;
	func_block.O3  :=	O3;
	func_block();
	Q0 := func_block.Q0;
	Q1 := func_block.Q1;
	Q2 := func_block.Q2;
	Q3 := func_block.Q3;

END_PROGRAM

CONFIGURATION Config0

	RESOURCE Res0 ON PLC
		TASK task0(INTERVAL := T#20ms,PRIORITY := 0);
		PROGRAM instance0 WITH task0 : program0;
	END_RESOURCE

END_CONFIGURATION

(* ---- SDT_TO_DATE.ST ---- *)
TYPE oscat_SDT :
	STRUCT
		YEAR : INT;
		MONTH : INT;
		DAY : INT;
		WEEKDAY : INT;
		HOUR : INT;
		MINUTE : INT;
		SECOND : INT;
		MS : INT;
	END_STRUCT;
END_TYPE

FUNCTION _INT_TO_UDINT:UDINT
	VAR_INPUT
		IN :	INT;
	END_VAR

	_INT_TO_UDINT := DINT_TO_UDINT(INT_TO_DINT(IN));
END_FUNCTION

FUNCTION SET_DATE:UDINT

	VAR_INPUT
		YEAR :	INT;
		MONTH :	INT;
		DAY :	INT;
	END_VAR

	VAR
		count :	INT;
	END_VAR

	IF month > 2 THEN
		count := (month - 1) * 30;
		IF month > 7 THEN
			count := count + DWORD_TO_INT(SHR(DINT_TO_DWORD(INT_TO_DINT(month) - INT_TO_DINT(3)),1));
		ELSE
			count := count + DWORD_TO_INT(SHR(DINT_TO_DWORD(INT_TO_DINT(month) - INT_TO_DINT(4)),1));
		END_IF;
		IF SHL(INT_TO_WORD(year),14) = WORD#0 THEN
			count := count + 1;
		END_IF;
	ELSE
		count := (month - 1) * 31;
	END_IF;
	SET_DATE := (_INT_TO_UDINT(count + day - 1) + DWORD_TO_UDINT(SHR(UDINT_TO_DWORD(_INT_TO_UDINT(year) * UDINT#1461 - UDINT#2878169), 2))) * UDINT#86400;

END_FUNCTION

FUNCTION_BLOCK SDT_TO_DATE_Block

	VAR_INPUT
		DTI :	oscat_SDT;
	END_VAR

	VAR_OUTPUT
		SDT_TO_DATE :	UDINT;
	END_VAR

	SDT_TO_DATE := SET_DATE(DTI.YEAR, DTI.MONTH, DTI.DAY);

END_FUNCTION_BLOCK

PROGRAM program0

	VAR
		DTI :	oscat_SDT;
		SDT_TO_DATE :	UDINT;
		func_block : SDT_TO_DATE_Block;
  	END_VAR
	func_block.DTI  :=	DTI;
	func_block();
	SDT_TO_DATE := func_block.SDT_TO_DATE;

END_PROGRAM

CONFIGURATION Config0

	RESOURCE Res0 ON PLC
		TASK task0(INTERVAL := T#20ms,PRIORITY := 0);
		PROGRAM instance0 WITH task0 : program0;
	END_RESOURCE

END_CONFIGURATION

(* ---- SDT_TO_DT.ST ---- *)
TYPE oscat_SDT :
	STRUCT
		YEAR : INT;
		MONTH : INT;
		DAY : INT;
		WEEKDAY : INT;
		HOUR : INT;
		MINUTE : INT;
		SECOND : INT;
		MS : INT;
	END_STRUCT;
END_TYPE

FUNCTION _INT_TO_UDINT:UDINT
	VAR_INPUT
		IN :	INT;
	END_VAR

	_INT_TO_UDINT := DINT_TO_UDINT(INT_TO_DINT(IN));
END_FUNCTION

FUNCTION SET_DATE:UDINT

	VAR_INPUT
		YEAR :	INT;
		MONTH :	INT;
		DAY :	INT;
	END_VAR

	VAR
		count :	INT;
	END_VAR

	IF month > 2 THEN
		count := (month - 1) * 30;
		IF month > 7 THEN
			count := count + DWORD_TO_INT(SHR(DINT_TO_DWORD(INT_TO_DINT(month) - INT_TO_DINT(3)),1));
		ELSE
			count := count + DWORD_TO_INT(SHR(DINT_TO_DWORD(INT_TO_DINT(month) - INT_TO_DINT(4)),1));
		END_IF;
		IF SHL(INT_TO_WORD(year),14) = WORD#0 THEN
			count := count + 1;
		END_IF;
	ELSE
		count := (month - 1) * 31;
	END_IF;
	SET_DATE := (_INT_TO_UDINT(count + day - 1) + DWORD_TO_UDINT(SHR(UDINT_TO_DWORD(_INT_TO_UDINT(year) * UDINT#1461 - UDINT#2878169), 2))) * UDINT#86400;

END_FUNCTION

FUNCTION SET_DT:UDINT
	VAR_INPUT
		YEAR :	INT;
		MONTH :	INT;
		DAY :	INT;
		HOUR :	INT;
		MINUTE :	INT;
		SECOND :	INT;
	END_VAR

	SET_DT := SET_DATE(YEAR, MONTH, DAY) + _INT_TO_UDINT(SECOND) + _INT_TO_UDINT(MINUTE) * UDINT#60 + _INT_TO_UDINT(HOUR) * UDINT#3600;
END_FUNCTION

FUNCTION_BLOCK SDT_TO_DT_Block

	VAR_INPUT
		DTI :	oscat_SDT;
	END_VAR

	VAR_OUTPUT
		SDT_TO_DT :	UDINT;
	END_VAR

	SDT_TO_DT := SET_DT(DTI.YEAR, DTI.MONTH, DTI.DAY, DTI.HOUR, DTI.MINUTE, DTI.SECOND);

END_FUNCTION_BLOCK

PROGRAM program0

	VAR
		DTI :	oscat_SDT;
		SDT_TO_DT :	UDINT;
		func_block : SDT_TO_DT_Block;
  	END_VAR
	func_block.DTI  :=	DTI;
	func_block();
	SDT_TO_DT := func_block.SDT_TO_DT;

END_PROGRAM

CONFIGURATION Config0

	RESOURCE Res0 ON PLC
		TASK task0(INTERVAL := T#20ms,PRIORITY := 0);
		PROGRAM instance0 WITH task0 : program0;
	END_RESOURCE

END_CONFIGURATION

(* ---- SDT_TO_TOD.ST ---- *)
TYPE oscat_SDT :
	STRUCT
		YEAR : INT;
		MONTH : INT;
		DAY : INT;
		WEEKDAY : INT;
		HOUR : INT;
		MINUTE : INT;
		SECOND : INT;
		MS : INT;
	END_STRUCT;
END_TYPE

FUNCTION _INT_TO_UDINT:UDINT
	VAR_INPUT
		IN :	INT;
	END_VAR

	_INT_TO_UDINT := DINT_TO_UDINT(INT_TO_DINT(IN));
END_FUNCTION

FUNCTION_BLOCK SDT_TO_TOD_Block

	VAR_INPUT
		DTI :	oscat_SDT;
	END_VAR

	VAR_OUTPUT
		SDT_TO_TOD :	UDINT;
	END_VAR

	SDT_TO_TOD := _INT_TO_UDINT(DTI.HOUR) * UDINT#3600000 + _INT_TO_UDINT(DTI.MINUTE) * UDINT#60000 + _INT_TO_UDINT(DTI.SECOND) * UDINT#1000 + _INT_TO_UDINT(DTI.MS);

END_FUNCTION_BLOCK

PROGRAM program0

	VAR
		DTI :	oscat_SDT;
		SDT_TO_TOD :	UDINT;
		func_block : SDT_TO_TOD_Block;
  	END_VAR
	func_block.DTI  :=	DTI;
	func_block();
	SDT_TO_TOD := func_block.SDT_TO_TOD;

END_PROGRAM

CONFIGURATION Config0

	RESOURCE Res0 ON PLC
		TASK task0(INTERVAL := T#20ms,PRIORITY := 0);
		PROGRAM instance0 WITH task0 : program0;
	END_RESOURCE

END_CONFIGURATION

(* ---- SEL2_OF_3.ST ---- *)
FUNCTION_BLOCK SEL2_OF_3_Block

	VAR_INPUT
		IN1 :	REAL;
		IN2 :	REAL;
		IN3 :	REAL;
		D :	REAL;
	END_VAR

	VAR_OUTPUT
		Y :	REAL;
		W :	INT;
		E :	BOOL;
	END_VAR

	VAR
		D12 :	BOOL;
		D23 :	BOOL;
		D31 :	BOOL;
	END_VAR

	D12 := ABS(IN1-IN2) <= D;
	D23 := ABS(IN2-IN3) <= D;
	D31 := ABS(IN3-IN1) <= D;

	IF (D12 AND D23) OR (D12 AND D31) OR (D23 AND D31) THEN
		Y := (IN1 + IN2 + IN3) * 0.333333333333;
		E := FALSE;
		W := 0;
	ELSIF D12 THEN
		Y := (In1 + IN2) * 0.5;
		E := FALSE;
		W := 3;
	ELSIF D23 THEN
		Y := (In2 + IN3) * 0.5;
		E := FALSE;
		W := 1;
	ELSIF D31 THEN
		Y := (In3 + IN1) * 0.5;
		E := FALSE;
		W := 2;
	ELSE
		E := TRUE;
		W := 4;
	END_IF;

END_FUNCTION_BLOCK

PROGRAM program0

	VAR
		IN1 :	REAL;
		IN2 :	REAL;
		IN3 :	REAL;
		D :	REAL;
		Y :	REAL;
		W :	INT;
		E :	BOOL;
		func_block : SEL2_OF_3_Block;
  	END_VAR
	func_block.IN1  :=IN1;
	func_block.IN2  :=IN2;
	func_block.IN3  :=IN3;
	func_block.D  :=D;
	func_block();
	Y := func_block.Y;
	W := func_block.W;
	E := func_block.E;

END_PROGRAM

CONFIGURATION Config0

	RESOURCE Res0 ON PLC
		TASK task0(INTERVAL := T#20ms,PRIORITY := 0);
		PROGRAM instance0 WITH task0 : program0;
	END_RESOURCE

END_CONFIGURATION

(* ---- SEL2_OF_3B.ST ---- *)
FUNCTION_BLOCK SEL2_OF_3B_Block

	VAR_INPUT
		IN1 :	BOOL;
		IN2 :	BOOL;
		IN3 :	BOOL;
		TD :	TIME;
	END_VAR

	VAR_OUTPUT
		Q :	BOOL;
		W :	BOOL;
	END_VAR

	VAR
		TDEL :	TON;
	END_VAR

	Q := (IN1 AND IN2) OR (IN1 AND IN3) OR (IN2 AND IN3);
	TDEL(IN := (in1 XOR in2) OR (in1 XOR in3) OR (in2 XOR in3), PT := TD);
	W := TDEL.Q;

END_FUNCTION_BLOCK

PROGRAM program0

	VAR
		IN1 :	BOOL;
		IN2 :	BOOL;
		IN3 :	BOOL;
		TD :	TIME;
		Q :	BOOL;
		W :	BOOL;
		func_block : SEL2_OF_3B_Block;
  	END_VAR
	func_block.IN1  :=IN1;
	func_block.IN2  :=IN2;
	func_block.IN3  :=IN3;
	func_block.TD  :=TD;
	func_block();
	Q := func_block.Q;
	W := func_block.W;

END_PROGRAM

CONFIGURATION Config0

	RESOURCE Res0 ON PLC
		TASK task0(INTERVAL := T#20ms,PRIORITY := 0);
		PROGRAM instance0 WITH task0 : program0;
	END_RESOURCE

END_CONFIGURATION

(* ---- SELECT_8.ST ---- *)
FUNCTION _BYTE_TO_INT:INT
	VAR_INPUT
		IN :	BYTE;
	END_VAR

	_BYTE_TO_INT := USINT_TO_INT(BYTE_TO_USINT(IN));
END_FUNCTION

FUNCTION INC:INT
	VAR_INPUT
		X :	INT;
		D :	INT;
		M :	INT;
	END_VAR

	inc := (X + D + M + 1) MOD (M + 1);
END_FUNCTION

FUNCTION_BLOCK SELECT_8_Block

	VAR_INPUT
		E :	BOOL;
		SET :	BOOL;
		IN :	BYTE;
		UP :	BOOL;
		DN :	BOOL;
		RST :	BOOL;
	END_VAR

	VAR_OUTPUT
		Q0 :	BOOL;
		Q1 :	BOOL;
		Q2 :	BOOL;
		Q3 :	BOOL;
		Q4 :	BOOL;
		Q5 :	BOOL;
		Q6 :	BOOL;
		Q7 :	BOOL;
		STATE :	INT;
	END_VAR

	VAR
		last_up :	BOOL;
		last_dn :	BOOL;
	END_VAR

	IF rst THEN
		state := 0;
	ELSIF set THEN
		state := _BYTE_TO_INT(IN);
	ELSIF up AND NOT last_up THEN
		state := inc(state,1,7);
	ELSIF dn AND NOT last_dn THEN
		state := inc(state,-1,7);
	END_IF;
	last_UP := UP;
	last_DN := DN;

	Q0 := FALSE;
	Q1 := FALSE;
	Q2 := FALSE;
	Q3 := FALSE;
	Q4 := FALSE;
	Q5 := FALSE;
	Q6 := FALSE;
	Q7 := FALSE;

	IF e THEN
		CASE state OF
			0: Q0 := TRUE;
			1: Q1 := TRUE;
			2: Q2 := TRUE;
			3: Q3 := TRUE;
			4: Q4 := TRUE;
			5: Q5 := TRUE;
			6: Q6 := TRUE;
			7: Q7 := TRUE;
		END_CASE;
	END_IF;

END_FUNCTION_BLOCK

PROGRAM program0
	VAR
		E :	BOOL;
		SET :	BOOL;
		IN :	BYTE;
		UP :	BOOL;
		DN :	BOOL;
		RST :	BOOL;
		Q0 :	BOOL;
		Q1 :	BOOL;
		Q2 :	BOOL;
		Q3 :	BOOL;
		Q4 :	BOOL;
		Q5 :	BOOL;
		Q6 :	BOOL;
		Q7 :	BOOL;
		STATE :	INT;
		func_block : SELECT_8_Block;
  	END_VAR
	func_block.E  :=E;
	func_block.SET  :=SET;
	func_block.IN  :=IN;
	func_block.UP  :=UP;
	func_block.DN  :=DN;
	func_block.RST  :=RST;
	func_block();
	Q0 := func_block.Q0;
	Q1 := func_block.Q1;
	Q2 := func_block.Q2;
	Q3 := func_block.Q3;
	Q4 := func_block.Q4;
	Q5 := func_block.Q5;
	Q6 := func_block.Q6;
	Q7 := func_block.Q7;
	STATE := func_block.STATE;
END_PROGRAM

CONFIGURATION Config0
	RESOURCE Res0 ON PLC
		TASK task0(INTERVAL := T#20ms,PRIORITY := 0);
		PROGRAM instance0 WITH task0 : program0;
	END_RESOURCE
END_CONFIGURATION

(* ---- SEQUENCE_4.ST ---- *)
FUNCTION UDINT_TO_TIME2:TIME

	VAR_INPUT
		IN :	UDINT;
	END_VAR

	UDINT_TO_TIME2 := DINT_TO_TIME(UDINT_TO_DINT(IN));

END_FUNCTION

FUNCTION_BLOCK T_PLC_MS_block
	VAR_OUTPUT
		T_PLC_MS :	UDINT;
	END_VAR

	VAR_EXTERNAL
		PLC_TICKS_PER_SEC :	INT;
		PLC_SYS_TICK_CNT :	DINT;
	END_VAR

	VAR
		debug :	BOOL;
		N :	INT;
		Offset :	UDINT;
		temp :	DWORD := DWORD#1;
		mode :	BOOL;
		faktor :	UDINT;
		init :	BOOL;
		v_plc_ticks_per_sec :	UDINT;
		base :	UDINT := UDINT#1000;
	END_VAR

	IF init = FALSE THEN
		v_plc_ticks_per_sec := INT_TO_UDINT(PLC_TICKS_PER_SEC);
		IF v_plc_ticks_per_sec = UDINT#1024 THEN
			faktor := UDINT#1;
			mode := FALSE;
		ELSIF v_plc_ticks_per_sec > UDINT#0 THEN
			IF v_plc_ticks_per_sec <= base THEN
				faktor := base / v_plc_ticks_per_sec;
				mode := FALSE;
			ELSE
				faktor := v_plc_ticks_per_sec / base;
				mode := TRUE;
			END_IF;
		ELSE
			faktor := UDINT#1;
		END_IF;
		init := TRUE;
	END_IF;

	IF mode THEN
		T_PLC_MS := DINT_TO_UDINT(PLC_SYS_TICK_CNT) / faktor;
	ELSE
		T_PLC_MS := DINT_TO_UDINT(PLC_SYS_TICK_CNT) * faktor;
	END_IF;

	IF debug THEN
		T_PLC_MS := (DWORD_TO_UDINT(SHL(UDINT_TO_DWORD(T_PLC_MS),N) OR SHL(temp,N)) - UDINT#1) + Offset;
	END_IF;

END_FUNCTION_BLOCK

FUNCTION_BLOCK SEQUENCE_4_Block

	VAR_INPUT
		IN0 :	BOOL := TRUE;
		IN1 :	BOOL := TRUE;
		IN2 :	BOOL := TRUE;
		IN3 :	BOOL := TRUE;
		START :	BOOL;
		RST :	BOOL;
		WAIT0 :	TIME;
		DELAY0 :	TIME;
		WAIT1 :	TIME;
		DELAY1 :	TIME;
		WAIT2 :	TIME;
		DELAY2 :	TIME;
		WAIT3 :	TIME;
		DELAY3 :	TIME;
		STOP_ON_ERROR :	BOOL;
	END_VAR

	VAR_OUTPUT
		Q0 :	BOOL;
		Q1 :	BOOL;
		Q2 :	BOOL;
		Q3 :	BOOL;
		QX :	BOOL;
		RUN :	BOOL;
		_STEP :	INT := -1;
		STATUS :	BYTE;
	END_VAR

	VAR
		last :	TIME;
		edge :	BOOL;
		tx :	TIME;
		init :	BOOL;
		T_PLC_MS :	T_PLC_MS_Block;
	END_VAR

	T_PLC_MS();
	tx:= UDINT_TO_TIME(T_PLC_MS.T_PLC_MS);

	IF NOT init THEN
		last := tx;
		init := TRUE;
		status := BYTE#110;
	END_IF;

	IF rst THEN
		_step := -1;
		Q0 := FALSE;
		Q1 := FALSE;
		Q2 := FALSE;
		Q3 := FALSE;
		status := BYTE#110;
		run := FALSE;

	ELSIF start AND NOT edge THEN
		_step := 0;
		last := tx;
		status := BYTE#111;
		Q0 := FALSE;
		Q1 := FALSE;
		Q2 := FALSE;
		Q3 := FALSE;
		run := TRUE;
	END_IF;
	edge := start;

	IF status > BYTE#0 AND status < BYTE#100 AND stop_on_error THEN RETURN; END_IF;

	IF run AND _step = 0 THEN
		IF NOT q0 AND in0 AND tx - last <= wait0 THEN
			Q0 := TRUE;
			last := tx;
		ELSIF NOT q0 AND tx - last > wait0 THEN
			status := BYTE#1;
			run := FALSE;
		ELSIF q0 AND tx - last >= delay0 THEN
			_step := 1;
			last := tx;
		END_IF;
	END_IF;
	IF run AND _step = 1 THEN
		IF NOT q1 AND in1 AND tx - last <= wait1 THEN
			Q0 := FALSE;
			Q1 := TRUE;
			last := tx;
		ELSIF NOT q1 AND Tx - last > wait1 THEN
			status := BYTE#2;
			q0 := FALSE;
			run := FALSE;
		ELSIF q1 AND tx - last >= delay1 THEN
			_step := 2;
			last := tx;
		END_IF;
	END_IF;
	IF run AND _step = 2 THEN
		IF NOT q2 AND in2 AND tx - last <= wait2 THEN
			Q1 := FALSE;
			Q2 := TRUE;
			last := tx;
		ELSIF NOT q2 AND Tx - last > wait2 THEN
			status := BYTE#3;
			q1 := FALSE;
			run := FALSE;
		ELSIF q2 AND tx - last >= delay2 THEN
			_step := 3;
			last := tx;
		END_IF;
	END_IF;
	IF run AND _step = 3 THEN
		IF NOT q3 AND in3 AND tx - last <= wait3 THEN
			Q2 := FALSE;
			Q3 := TRUE;
			last := tx;
		ELSIF NOT q3 AND Tx - last > wait3 THEN
			status := BYTE#4;
			q2 := FALSE;
			run := FALSE;
		ELSIF q3 AND tx - last >= delay3 THEN
			_step := -1;
			q3 := FALSE;
			run := FALSE;
			status := BYTE#110;
		END_IF;
	END_IF;
	QX := q0 OR q1 OR q2 OR q3;

END_FUNCTION_BLOCK

PROGRAM program0

	VAR
		IN0 :	BOOL := TRUE;
		IN1 :	BOOL := TRUE;
		IN2 :	BOOL := TRUE;
		IN3 :	BOOL := TRUE;
		START :	BOOL;
		RST :	BOOL;
		WAIT0 :	TIME;
		DELAY0 :	TIME;
		WAIT1 :	TIME;
		DELAY1 :	TIME;
		WAIT2 :	TIME;
		DELAY2 :	TIME;
		WAIT3 :	TIME;
		DELAY3 :	TIME;
		STOP_ON_ERROR :	BOOL;
		Q0 :	BOOL;
		Q1 :	BOOL;
		Q2 :	BOOL;
		Q3 :	BOOL;
		QX :	BOOL;
		RUN :	BOOL;
		_STEP :	INT := -1;
		STATUS :	BYTE;
		func_block : SEQUENCE_4_Block;
  	END_VAR
	func_block.IN0  :=IN0;
	func_block.IN1  :=IN1;
	func_block.IN2  :=IN2;
	func_block.IN3  :=IN3;
	func_block.START  :=START;
	func_block.RST  :=RST;
	func_block.WAIT0  :=WAIT0;
	func_block.DELAY0  :=DELAY0;
	func_block.WAIT1:=WAIT1;
	func_block.DELAY1:=DELAY1;
	func_block.WAIT2  :=WAIT2;
	func_block.DELAY2  :=DELAY2;
	func_block.WAIT3  :=WAIT3;
	func_block.DELAY3  :=DELAY3;
	func_block.DELAY1:=DELAY1;
	func_block.WAIT2  :=WAIT2;
	func_block.DELAY2  :=DELAY2;
	func_block.WAIT3  :=WAIT3;
	func_block.DELAY3  :=DELAY3;
	func_block.STOP_ON_ERROR  :=STOP_ON_ERROR;
	func_block();
	Q0 := func_block.Q0;
	Q1 := func_block.Q1;
	Q2 := func_block.Q2;
	Q3 := func_block.Q3;
	QX := func_block.QX;
	RUN := func_block.RUN;
	_STEP := func_block._STEP;
	STATUS := func_block.STATUS;

END_PROGRAM

CONFIGURATION Config0

	VAR_GLOBAL
		PLC_TICKS_PER_SEC :	INT;
		PLC_SYS_TICK_CNT :	DINT;
	END_VAR

	RESOURCE Res0 ON PLC
		TASK task0(INTERVAL := T#20ms,PRIORITY := 0);
		PROGRAM instance0 WITH task0 : program0;
	END_RESOURCE

END_CONFIGURATION

(* ---- SEQUENCE_64.ST ---- *)
TYPE
	oscat_array64_time          : ARRAY [0..63]   OF TIME;
END_TYPE

FUNCTION INC2:INT

	VAR_INPUT
		X :	INT;
		D :	INT;
		L :	INT;
		U :	INT;
	END_VAR

	VAR
		tmp :	INT;
	END_VAR

	tmp := U - L + 1;
	INC2 := (X + D - L + tmp) MOD tmp + L;

END_FUNCTION

FUNCTION UDINT_TO_TIME2:TIME

	VAR_INPUT
		IN :	UDINT;
	END_VAR

	UDINT_TO_TIME2 := DINT_TO_TIME(UDINT_TO_DINT(IN));

END_FUNCTION

FUNCTION_BLOCK T_PLC_MS_block
	VAR_OUTPUT
		T_PLC_MS :	UDINT;
	END_VAR

	VAR_EXTERNAL
		PLC_TICKS_PER_SEC :	INT;
		PLC_SYS_TICK_CNT :	DINT;
	END_VAR

	VAR
		debug :	BOOL;(*Debug-Mode ON / OFF*)
		N :	INT;(*Debug-Faktor*)
		Offset :	UDINT;(*Debug-Offset*)
		temp :	DWORD := DWORD#1;(*Debug-Offset*)
		mode :	BOOL;(*modus*)
		faktor :	UDINT;(*Systemtakt-Faktor*)
		init :	BOOL;
		v_plc_ticks_per_sec :	UDINT;
		base :	UDINT := UDINT#1000;
	END_VAR

	IF init = FALSE THEN
		v_plc_ticks_per_sec := INT_TO_UDINT(PLC_TICKS_PER_SEC);
		IF v_plc_ticks_per_sec = UDINT#1024 THEN
			faktor := UDINT#1;
			mode := FALSE;
		ELSIF v_plc_ticks_per_sec > UDINT#0 THEN
			IF v_plc_ticks_per_sec <= base THEN
				faktor := base / v_plc_ticks_per_sec;
				mode := FALSE;
			ELSE
				faktor := v_plc_ticks_per_sec / base;
				mode := TRUE;
			END_IF;
		ELSE
			faktor := UDINT#1;
		END_IF;
		init := TRUE;
	END_IF;

	IF mode THEN
		T_PLC_MS := DINT_TO_UDINT(PLC_SYS_TICK_CNT) / faktor;
	ELSE
		T_PLC_MS := DINT_TO_UDINT(PLC_SYS_TICK_CNT) * faktor;
	END_IF;

	IF debug THEN
		T_PLC_MS := (DWORD_TO_UDINT(SHL(UDINT_TO_DWORD(T_PLC_MS),N) OR SHL(temp,N)) - UDINT#1) + Offset;
	END_IF;

END_FUNCTION_BLOCK

FUNCTION_BLOCK SEQUENCE_64_Block

	VAR_INPUT
		START :	BOOL;
		SMAX :	INT;
		RST :	BOOL;
	END_VAR

	VAR_OUTPUT
		STATE :	INT := INT#-1;
		TRIG :	BOOL;
	END_VAR

	VAR_IN_OUT
		PROG :	oscat_array64_time;
	END_VAR

	VAR
		T_PLC_MS :	T_PLC_MS_block;
		tx :	TIME;
		last :	TIME;
		edge :	BOOL;
	END_VAR

	T_PLC_MS();
	tx:= UDINT_TO_TIME(T_PLC_MS.T_PLC_MS);
	TRIG := FALSE;

	IF RST THEN
		STATE := -1;

	ELSIF START AND NOT edge THEN
		STATE := 0;
		last := tx;
		TRIG := TRUE;

	ELSIF (STATE >= 0) THEN
		IF (tx - last) >= PROG[STATE] THEN
			STATE := INC2(STATE, 1, -1, SMAX);
			last := tx;
			TRIG := TRUE;
		END_IF;
	END_IF;

	edge := START;
END_FUNCTION_BLOCK

PROGRAM program0
	VAR
		START :	BOOL;
		SMAX :	INT;
		RST :	BOOL;
		STATE :	INT := INT#-1;
		TRIG :	BOOL;
		func_block : SEQUENCE_64_Block;
  	END_VAR
	func_block.START  :=START;
	func_block.SMAX  :=SMAX;
	func_block.RST  :=RST;
	func_block();
	STATE := func_block.STATE;
	TRIG := func_block.TRIG;
END_PROGRAM

CONFIGURATION Config0

	VAR_GLOBAL
		PLC_TICKS_PER_SEC :	INT;
		PLC_SYS_TICK_CNT :	DINT;
	END_VAR

  	RESOURCE Res0 ON PLC
    	TASK task0(INTERVAL := T#20ms,PRIORITY := 0);
    	PROGRAM instance0 WITH task0 : program0;
  	END_RESOURCE

END_CONFIGURATION

(* ---- SEQUENCE_8.ST ---- *)
FUNCTION UDINT_TO_TIME2:TIME

	VAR_INPUT
		IN :	UDINT;
	END_VAR

	UDINT_TO_TIME2 := DINT_TO_TIME(UDINT_TO_DINT(IN));

END_FUNCTION

FUNCTION_BLOCK T_PLC_MS_block
	VAR_OUTPUT
		T_PLC_MS :	UDINT;
	END_VAR

	VAR_EXTERNAL
		PLC_TICKS_PER_SEC :	INT;
		PLC_SYS_TICK_CNT :	DINT;
	END_VAR

	VAR
		debug :	BOOL;
		N :	INT;
		Offset :	UDINT;
		temp :	DWORD := DWORD#1;
		mode :	BOOL;
		faktor :	UDINT;
		init :	BOOL;
		v_plc_ticks_per_sec :	UDINT;
		base :	UDINT := UDINT#1000;
	END_VAR

	IF init = FALSE THEN
		v_plc_ticks_per_sec := INT_TO_UDINT(PLC_TICKS_PER_SEC);
		IF v_plc_ticks_per_sec = UDINT#1024 THEN
			faktor := UDINT#1;
			mode := FALSE;
		ELSIF v_plc_ticks_per_sec > UDINT#0 THEN
			IF v_plc_ticks_per_sec <= base THEN
				faktor := base / v_plc_ticks_per_sec;
				mode := FALSE;
			ELSE
				faktor := v_plc_ticks_per_sec / base;
				mode := TRUE;
			END_IF;
		ELSE
			faktor := UDINT#1;
		END_IF;
		init := TRUE;
	END_IF;

	IF mode THEN
		T_PLC_MS := DINT_TO_UDINT(PLC_SYS_TICK_CNT) / faktor;
	ELSE
		T_PLC_MS := DINT_TO_UDINT(PLC_SYS_TICK_CNT) * faktor;
	END_IF;

	IF debug THEN
		T_PLC_MS := (DWORD_TO_UDINT(SHL(UDINT_TO_DWORD(T_PLC_MS),N) OR SHL(temp,N)) - UDINT#1) + Offset;
	END_IF;

END_FUNCTION_BLOCK

FUNCTION_BLOCK SEQUENCE_8_Block

	VAR_INPUT
		IN0 :	BOOL := TRUE;
		IN1 :	BOOL := TRUE;
		IN2 :	BOOL := TRUE;
		IN3 :	BOOL := TRUE;
		IN4 :	BOOL := TRUE;
		IN5 :	BOOL := TRUE;
		IN6 :	BOOL := TRUE;
		IN7 :	BOOL := TRUE;
		START :	BOOL;
		RST :	BOOL;
		WAIT0 :	TIME;
		DELAY0 :	TIME;
		WAIT1 :	TIME;
		DELAY1 :	TIME;
		WAIT2 :	TIME;
		DELAY2 :	TIME;
		WAIT3 :	TIME;
		DELAY3 :	TIME;
		WAIT4 :	TIME;
		DELAY4 :	TIME;
		WAIT5 :	TIME;
		DELAY5 :	TIME;
		WAIT6 :	TIME;
		DELAY6 :	TIME;
		WAIT7 :	TIME;
		DELAY7 :	TIME;
		STOP_ON_ERROR :	BOOL;
	END_VAR

	VAR_OUTPUT
		Q0 :	BOOL;
		Q1 :	BOOL;
		Q2 :	BOOL;
		Q3 :	BOOL;
		Q4 :	BOOL;
		Q5 :	BOOL;
		Q6 :	BOOL;
		Q7 :	BOOL;
		QX :	BOOL;
		RUN :	BOOL;
		_STEP :	INT := -1;
		STATUS :	BYTE;
	END_VAR

	VAR
		last :	TIME;
		edge :	BOOL;
		tx :	TIME;
		init :	BOOL;
		T_PLC_MS :	T_PLC_MS_Block;
	END_VAR

	T_PLC_MS();
	tx:= UDINT_TO_TIME(T_PLC_MS.T_PLC_MS);

	IF NOT init THEN
		last := tx;
		init := TRUE;
		status := BYTE#110;
	END_IF;

	IF rst THEN
		_step := -1;
		Q0 := FALSE;
		Q1 := FALSE;
		Q2 := FALSE;
		Q3 := FALSE;
		Q4 := FALSE;
		Q5 := FALSE;
		Q6 := FALSE;
		Q7 := FALSE;
		status := BYTE#110;
		run := FALSE;

	ELSIF start AND NOT edge THEN
		_step := 0;
		last := tx;
		status := BYTE#111;
		Q0 := FALSE;
		Q1 := FALSE;
		Q2 := FALSE;
		Q3 := FALSE;
		Q4 := FALSE;
		Q5 := FALSE;
		Q6 := FALSE;
		Q7 := FALSE;
		run := TRUE;
	END_IF;
	edge := start;

	IF status > BYTE#0 AND status < BYTE#100 AND stop_on_error THEN RETURN; END_IF;

	IF run AND _step = 0 THEN
		IF NOT q0 AND in0 AND tx - last <= wait0 THEN
			Q0 := TRUE;
			last := tx;
		ELSIF NOT q0 AND tx - last > wait0 THEN
			status := BYTE#1;
			run := FALSE;
		ELSIF q0 AND tx - last >= delay0 THEN
			_step := 1;
			last := tx;
		END_IF;
	END_IF;
	IF run AND _step = 1 THEN
		IF NOT q1 AND in1 AND tx - last <= wait1 THEN
			Q0 := FALSE;
			Q1 := TRUE;
			last := tx;
		ELSIF NOT q1 AND Tx - last > wait1 THEN
			status := BYTE#2;
			q0 := FALSE;
			run := FALSE;
		ELSIF q1 AND tx - last >= delay1 THEN
			_step := 2;
			last := tx;
		END_IF;
	END_IF;
	IF run AND _step = 2 THEN
		IF NOT q2 AND in2 AND tx - last <= wait2 THEN
			Q1 := FALSE;
			Q2 := TRUE;
			last := tx;
		ELSIF NOT q2 AND Tx - last > wait2 THEN
			status := BYTE#3;
			q1 := FALSE;
			run := FALSE;
		ELSIF q2 AND tx - last >= delay2 THEN
			_step := 3;
			last := tx;
		END_IF;
	END_IF;
	IF run AND _step = 3 THEN
		IF NOT q3 AND in3 AND tx - last <= wait3 THEN
			Q2 := FALSE;
			Q3 := TRUE;
			last := tx;
		ELSIF NOT q3 AND Tx - last > wait3 THEN
			status := BYTE#4;
			q2 := FALSE;
			run := FALSE;
		ELSIF q3 AND tx - last >= delay3 THEN
			_step := 4;
			last := tx;
		END_IF;
	END_IF;
	IF run AND _step = 4 THEN
		IF NOT q4 AND in4 AND tx - last <= wait4 THEN
			Q3 := FALSE;
			Q4 := TRUE;
			last := tx;
		ELSIF NOT q4 AND Tx - last > wait4 THEN
			status := BYTE#5;
			q3 := FALSE;
			run := FALSE;
		ELSIF q4 AND tx - last >= delay4 THEN
			_step := 5;
			last := tx;
		END_IF;
	END_IF;
	IF run AND _step = 5 THEN
		IF NOT q5 AND in5 AND tx - last <= wait5 THEN
			Q4 := FALSE;
			Q5 := TRUE;
			last := tx;
		ELSIF NOT q5 AND Tx - last > wait5 THEN
			status := BYTE#6;
			q4 := FALSE;
			run := FALSE;
		ELSIF q5 AND tx - last >= delay5 THEN
			_step := 6;
			last := tx;
		END_IF;
	END_IF;
	IF run AND _step = 6 THEN
		IF NOT q6 AND in6 AND tx - last <= wait6 THEN
			Q5 := FALSE;
			Q6 := TRUE;
			last := tx;
		ELSIF NOT q6 AND Tx - last > wait6 THEN
			status := BYTE#7;
			q5 := FALSE;
			run := FALSE;
		ELSIF q6 AND tx - last >= delay6 THEN
			_step := 7;
			last := tx;
		END_IF;
	END_IF;
	IF run AND _step = 7 THEN
		IF NOT q7 AND in7 AND tx - last <= wait7 THEN
			Q6 := FALSE;
			Q7 := TRUE;
			last := tx;
		ELSIF NOT q7 AND Tx - last > wait7 THEN
			status := BYTE#8;
			q6 := FALSE;
			run := FALSE;
		ELSIF q7 AND tx - last >= delay7 THEN
			_step := -1;
			Q7 := FALSE;
			Run := FALSE;
			status := BYTE#110;
		END_IF;
	END_IF;
	QX := q0 OR q1 OR q2 OR q3 OR q4 OR q5 OR q6 OR q7;

END_FUNCTION_BLOCK

PROGRAM program0

	VAR
		IN0 :	BOOL := TRUE;
		IN1 :	BOOL := TRUE;
		IN2 :	BOOL := TRUE;
		IN3 :	BOOL := TRUE;
		IN4 :	BOOL := TRUE;
		IN5 :	BOOL := TRUE;
		IN6 :	BOOL := TRUE;
		IN7 :	BOOL := TRUE;
		START :	BOOL;
		RST :	BOOL;
		WAIT0 :	TIME;
		DELAY0 :	TIME;
		WAIT1 :	TIME;
		DELAY1 :	TIME;
		WAIT2 :	TIME;
		DELAY2 :	TIME;
		WAIT3 :	TIME;
		DELAY3 :	TIME;
		WAIT4 :	TIME;
		DELAY4 :	TIME;
		WAIT5 :	TIME;
		DELAY5 :	TIME;
		WAIT6 :	TIME;
		DELAY6 :	TIME;
		WAIT7 :	TIME;
		DELAY7 :	TIME;
		STOP_ON_ERROR :	BOOL;
		Q0 :	BOOL;
		Q1 :	BOOL;
		Q2 :	BOOL;
		Q3 :	BOOL;
		Q4 :	BOOL;
		Q5 :	BOOL;
		Q6 :	BOOL;
		Q7 :	BOOL;
		QX :	BOOL;
		RUN :	BOOL;
		_STEP :	INT := -1;
		STATUS :	BYTE;
		func_block : SEQUENCE_8_Block;
  	END_VAR
	func_block.IN0  :=IN0;
	func_block.IN1  :=IN1;
	func_block.IN2  :=IN2;
	func_block.IN3  :=IN3;
	func_block.IN4  :=IN4;
	func_block.IN5  :=IN5;
	func_block.IN6  :=IN6;
	func_block.IN7  :=IN7;
	func_block.START  :=START;
	func_block.RST  :=RST;
	func_block.WAIT0  :=WAIT0;
	func_block.DELAY0  :=DELAY0;
	func_block.WAIT1:=WAIT1;
	func_block.DELAY1:=DELAY1;
	func_block.WAIT2  :=WAIT2;
	func_block.DELAY2  :=DELAY2;
	func_block.WAIT3  :=WAIT3;
	func_block.DELAY3  :=DELAY3;
	func_block.DELAY1:=DELAY1;
	func_block.WAIT2  :=WAIT2;
	func_block.DELAY2  :=DELAY2;
	func_block.WAIT3  :=WAIT3;
	func_block.DELAY3  :=DELAY3;
	func_block.WAIT4:=WAIT4;
	func_block.DELAY4  :=DELAY4;
	func_block.WAIT5  :=WAIT5;
	func_block.DELAY5  :=DELAY5;
	func_block.WAIT6  :=WAIT6;
	func_block.DELAY6  :=DELAY6;
	func_block.WAIT7  :=WAIT7;
	func_block.DELAY7  :=DELAY7;
	func_block.STOP_ON_ERROR  :=STOP_ON_ERROR;
	func_block();
	Q0 := func_block.Q0;
	Q1 := func_block.Q1;
	Q2 := func_block.Q2;
	Q3 := func_block.Q3;
	Q4 := func_block.Q4;
	Q5 := func_block.Q5;
	Q6 := func_block.Q6;
	Q7 := func_block.Q7;
	QX := func_block.QX;
	RUN := func_block.RUN;
	_STEP := func_block._STEP;
	STATUS := func_block.STATUS;

END_PROGRAM

CONFIGURATION Config0

	VAR_GLOBAL
		PLC_TICKS_PER_SEC :	INT;
		PLC_SYS_TICK_CNT :	DINT;
	END_VAR

	RESOURCE Res0 ON PLC
		TASK task0(INTERVAL := T#20ms,PRIORITY := 0);
		PROGRAM instance0 WITH task0 : program0;
	END_RESOURCE

END_CONFIGURATION

(* ---- SETUP_CHARNAMES.ST ---- *)
TYPE
  oscat_CHARNAMES	: ARRAY [1..11] OF STRING;
END_TYPE

FUNCTION_BLOCK SETUP_CHARNAMES_Block

	VAR_IN_OUT
		CHARNAMES :	oscat_CHARNAMES;
	END_VAR

	VAR
		init :	BOOL;
	END_VAR

	IF init THEN RETURN; END_IF;

	init := TRUE;

	CHARNAMES[01] := '123';
	CHARNAMES[02] := '456';
	CHARNAMES[03] := 'zgsdafasf';
	CHARNAMES[04] := 'sadfsdfa';
	CHARNAMES[05] := 'asdfdsafdfds';
	CHARNAMES[06] := 'sadfsdfsdf';
	CHARNAMES[07] := 'sfsfdfdddd';
	CHARNAMES[08] := 'dddddted';
	CHARNAMES[10] := 'wer';
	CHARNAMES[11] := 'werwer';

END_FUNCTION_BLOCK

PROGRAM program0

	VAR
		CHARNAMES :	oscat_CHARNAMES;
		func_block : SETUP_CHARNAMES_Block;
  	END_VAR
	func_block.CHARNAMES  :=CHARNAMES;
	func_block();
	CHARNAMES := func_block.CHARNAMES;

END_PROGRAM

CONFIGURATION Config0

	RESOURCE Res0 ON PLC
		TASK task0(INTERVAL := T#20ms,PRIORITY := 0);
		PROGRAM instance0 WITH task0 : program0;
	END_RESOURCE

END_CONFIGURATION

(* ---- SETUP_DIRS.ST ---- *)
TYPE
  oscat_ELEMENT_DIRS 		: ARRAY [0..15] OF STRING;
  oscat_DIRS				: ARRAY [1..3]  OF oscat_ELEMENT_DIRS := [0,0 , 0];
END_TYPE

FUNCTION_BLOCK SETUP_DIRS
	VAR_IN_OUT
		DIRS :	oscat_DIRS;
	END_VAR

	VAR
		init :	BOOL;
	END_VAR

	IF init THEN RETURN; END_IF;
	init := TRUE;

	(* ---- english --- *)
	DIRS[1][00] := 'N';
	DIRS[1][01] := 'NNE';
	DIRS[1][02] := 'NE';
	DIRS[1][03] := 'ENE';
	DIRS[1][04] := 'E';
	DIRS[1][05] := 'ESE';
	DIRS[1][06] := 'SE';
	DIRS[1][07] := 'SSE';
	DIRS[1][08] := 'S';
	DIRS[1][09] := 'SSW';
	DIRS[1][10] := 'SW';
	DIRS[1][11] := 'WSW';
	DIRS[1][12] := 'W';
	DIRS[1][13] := 'WNW';
	DIRS[1][14] := 'NW';
	DIRS[1][15] := 'NNW';

	(* ---- german --- *)
	DIRS[2][00] := 'N';
	DIRS[2][01] := 'NNO';
	DIRS[2][02] := 'NO';
	DIRS[2][03] := 'ONO';
	DIRS[2][04] := 'O';
	DIRS[2][05] := 'OSO';
	DIRS[2][06] := 'SO';
	DIRS[2][07] := 'SSO';
	DIRS[2][08] := 'S';
	DIRS[2][09] := 'SSW';
	DIRS[2][10] := 'SW';
	DIRS[2][11] := 'WSW';
	DIRS[2][12] := 'W';
	DIRS[2][13] := 'WNW';
	DIRS[2][14] := 'NW';
	DIRS[2][15] := 'NNW';

	(* ---- french --- *)
	DIRS[3][00] := 'N';
	DIRS[3][01] := 'NNO';
	DIRS[3][02] := 'NO';
	DIRS[3][03] := 'ONO';
	DIRS[3][04] := 'O';
	DIRS[3][05] := 'OSO';
	DIRS[3][06] := 'SO';
	DIRS[3][07] := 'SSO';
	DIRS[3][08] := 'S';
	DIRS[3][09] := 'SSW';
	DIRS[3][10] := 'SW';
	DIRS[3][11] := 'WSW';
	DIRS[3][12] := 'W';
	DIRS[3][13] := 'WNW';
	DIRS[3][14] := 'NW';
	DIRS[3][15] := 'NNW';
END_FUNCTION_BLOCK

PROGRAM program0
  VAR
    LocalVar0 : oscat_DIRS;
	LocalOUT  : BOOL;
	func_block : SETUP_DIRS;
  END_VAR
	func_block.DIRS  := LocalVar0;
	func_block();
	LocalOUT := func_block.init;
END_PROGRAM

CONFIGURATION Config0
  RESOURCE Res0 ON PLC
    TASK task0(INTERVAL := T#20ms,PRIORITY := 0);
    PROGRAM instance0 WITH task0 : program0;
  END_RESOURCE
END_CONFIGURATION

(* ---- SETUP_HOLIDAY_AT.ST ---- *)
TYPE oscat_HOLIDAY_DATA :
	STRUCT
		NAME : STRING;
		DAY : SINT;
		MONTH : SINT;
		USE : SINT;
		PAD_BYTE : BYTE;
	END_STRUCT;
END_TYPE

TYPE
	oscat_HOLIDAY_DATA_0_29 	: ARRAY [0..29] OF oscat_HOLIDAY_DATA;
END_TYPE

FUNCTION_BLOCK SETUP_HOLIDAY_AT_Block

	VAR_IN_OUT
		HD :	oscat_HOLIDAY_DATA_0_29;
	END_VAR

	VAR
		init :	BOOL;
	END_VAR

	IF init THEN RETURN; END_IF;

	init := TRUE;

	HD[00].NAME := 'Neujahr';
	HD[00].DAY  := SINT#01;
	HD[00].MONTH := SINT#01;
	HD[00].USE := SINT#01;

	HD[01].NAME := 'Heilige Drei Koenige';
	HD[01].DAY  := SINT#06;
	HD[01].MONTH := SINT#01;
	HD[01].USE := SINT#01;

	HD[02].NAME := 'Karfreitag';
	HD[02].DAY  := SINT#-2;
	HD[02].MONTH := SINT#00;
	HD[02].USE := SINT#01;

	HD[03].NAME := 'Ostersonntag';
	HD[03].DAY  := SINT#00;
	HD[03].MONTH := SINT#00;
	HD[03].USE := SINT#01;

	HD[04].NAME := 'Ostermontag';
	HD[04].DAY  := SINT#01;
	HD[04].MONTH := SINT#00;
	HD[04].USE := SINT#01;

	HD[05].NAME := '';
	HD[05].DAY  := SINT#01;
	HD[05].MONTH := SINT#05;
	HD[05].USE := SINT#00;

	HD[06].NAME := 'Christi Himmelfahrt';
	HD[06].DAY  := SINT#39;
	HD[06].MONTH := SINT#00;
	HD[06].USE := SINT#01;

	HD[07].NAME := 'Pfingstsonntag';
	HD[07].DAY  := SINT#49;
	HD[07].MONTH := SINT#00;
	HD[07].USE := SINT#01;

	HD[08].NAME := 'Pfingstmontag';
	HD[08].DAY  := SINT#50;
	HD[08].MONTH := SINT#00;
	HD[08].USE := SINT#01;

	HD[09].NAME := 'Fronleichnam';
	HD[09].DAY  := SINT#60;
	HD[09].MONTH := SINT#00;
	HD[09].USE := SINT#01;

	HD[10].NAME := '';
	HD[10].DAY  := SINT#08;
	HD[10].MONTH := SINT#08;
	HD[10].USE := SINT#00;

	HD[11].NAME := 'Maria Himmelfahrt';
	HD[11].DAY  := SINT#15;
	HD[11].MONTH := SINT#08;
	HD[11].USE := SINT#01;

	HD[12].NAME := '';
	HD[12].DAY  := SINT#03;
	HD[12].MONTH := SINT#10;
	HD[12].USE := SINT#00;

	HD[13].NAME := '';
	HD[13].DAY  := SINT#31;
	HD[13].MONTH := SINT#10;
	HD[13].USE := SINT#00;

	HD[14].NAME := 'Allerheiligen';
	HD[14].DAY  := SINT#01;
	HD[14].MONTH := SINT#11;
	HD[14].USE := SINT#01;

	HD[15].NAME := 'Maria Empfngnis';
	HD[15].DAY  := SINT#8;
	HD[15].MONTH := SINT#12;
	HD[15].USE := SINT#01;

	HD[16].NAME := '1. Weihnachtsfeiertag';
	HD[16].DAY  := SINT#25;
	HD[16].MONTH := SINT#12;
	HD[16].USE := SINT#01;

	HD[17].NAME := '2. Weihnachtsfeiertag';
	HD[17].DAY  := SINT#26;
	HD[17].MONTH := SINT#12;
	HD[17].USE := SINT#01;

END_FUNCTION_BLOCK

PROGRAM program0

	VAR
		LocalVar0 : oscat_HOLIDAY_DATA_0_29;
		func_block : SETUP_HOLIDAY_AT_Block;
	END_VAR
		func_block.HD  := LocalVar0;
		func_block();
		LocalVar0 := func_block.HD;

END_PROGRAM

CONFIGURATION Config0

	RESOURCE Res0 ON PLC
		TASK task0(INTERVAL := T#20ms,PRIORITY := 0);
		PROGRAM instance0 WITH task0 : program0;
	END_RESOURCE

END_CONFIGURATION

(* ---- SETUP_HOLIDAY_DE.ST ---- *)
TYPE oscat_HOLIDAY_DATA :
	STRUCT
		NAME : STRING;
		DAY : SINT;
		MONTH : SINT;
		USE : SINT;
		PAD_BYTE : BYTE;
	END_STRUCT;
END_TYPE

TYPE
	oscat_HOLIDAY_DATA_0_29 	: ARRAY [0..29] OF oscat_HOLIDAY_DATA;
END_TYPE

FUNCTION_BLOCK SETUP_HOLIDAY_DE_Block

	VAR_IN_OUT
		HD :	oscat_HOLIDAY_DATA_0_29;
	END_VAR

	VAR
		init :	BOOL;
	END_VAR

	IF init THEN RETURN; END_IF;

	init := TRUE;

	(* ---- german --- *)

	HD[00].NAME := 'Neujahr';
	HD[00].DAY  := SINT#01;
	HD[00].MONTH := SINT#01;
	HD[00].USE := SINT#01;

	HD[01].NAME := 'Heilige Drei Koenige';
	HD[01].DAY  := SINT#06;
	HD[01].MONTH := SINT#01;
	HD[01].USE := SINT#01;

	HD[02].NAME := 'Karfreitag';
	HD[02].DAY  := SINT#-2;
	HD[02].MONTH := SINT#00;
	HD[02].USE := SINT#01;

	HD[03].NAME := 'Ostersonntag';
	HD[03].DAY  := SINT#00;
	HD[03].MONTH := SINT#00;
	HD[03].USE := SINT#01;

	HD[04].NAME := 'Ostermontag';
	HD[04].DAY  := SINT#01;
	HD[04].MONTH := SINT#00;
	HD[04].USE := SINT#01;

	HD[05].NAME := 'Tag der Arbeit';
	HD[05].DAY  := SINT#01;
	HD[05].MONTH := SINT#05;
	HD[05].USE := SINT#01;

	HD[06].NAME := 'Christi Himmelfahrt';
	HD[06].DAY  := SINT#39;
	HD[06].MONTH := SINT#00;
	HD[06].USE := SINT#01;

	HD[07].NAME := 'Pfingstsonntag';
	HD[07].DAY  := SINT#49;
	HD[07].MONTH := SINT#00;
	HD[07].USE := SINT#01;

	HD[08].NAME := 'Pfingstmontag';
	HD[08].DAY  := SINT#50;
	HD[08].MONTH := SINT#00;
	HD[08].USE := SINT#01;

	HD[09].NAME := 'Fronleichnam';
	HD[09].DAY  := SINT#60;
	HD[09].MONTH := SINT#00;
	HD[09].USE := SINT#01;

	HD[10].NAME := 'Augsburger Friedensfest';
	HD[10].DAY  := SINT#08;
	HD[10].MONTH := SINT#08;
	HD[10].USE := SINT#00;

	HD[11].NAME := 'Maria Himmelfahrt';
	HD[11].DAY  := SINT#15;
	HD[11].MONTH := SINT#08;
	HD[11].USE := SINT#01;

	HD[12].NAME := 'Tag der Deutschen Einheit';
	HD[12].DAY  := SINT#03;
	HD[12].MONTH := SINT#10;
	HD[12].USE := SINT#01;

	HD[13].NAME := 'Reformationstag';
	HD[13].DAY  := SINT#31;
	HD[13].MONTH := SINT#10;
	HD[13].USE := SINT#00;

	HD[14].NAME := 'Allerheiligen';
	HD[14].DAY  := SINT#01;
	HD[14].MONTH := SINT#11;
	HD[14].USE := SINT#01;

	HD[15].NAME := 'Buss und Bettag';
	HD[15].DAY  := SINT#23;
	HD[15].MONTH := SINT#11;
	HD[15].USE := SINT#00;

	HD[16].NAME := '1. Weihnachtsfeiertag';
	HD[16].DAY  := SINT#25;
	HD[16].MONTH := SINT#12;
	HD[16].USE := SINT#01;

	HD[17].NAME := '2. Weihnachtsfeiertag';
	HD[17].DAY  := SINT#26;
	HD[17].MONTH := SINT#12;
	HD[17].USE := SINT#01;

END_FUNCTION_BLOCK

PROGRAM program0
	VAR
		LocalVar0 : oscat_HOLIDAY_DATA_0_29;
		func_block : SETUP_HOLIDAY_DE_Block;
	END_VAR
		func_block.HD  := LocalVar0;
		func_block();
		LocalVar0 := func_block.HD;
END_PROGRAM

CONFIGURATION Config0
	RESOURCE Res0 ON PLC
		TASK task0(INTERVAL := T#20ms,PRIORITY := 0);
		PROGRAM instance0 WITH task0 : program0;
	END_RESOURCE
END_CONFIGURATION

(* ---- SETUP_HOLIDAY_FR.ST ---- *)
TYPE oscat_HOLIDAY_DATA :
	STRUCT
		NAME : STRING;
		DAY : SINT;
		MONTH : SINT;
		USE : SINT;
		PAD_BYTE : BYTE;
	END_STRUCT;
END_TYPE

TYPE
	oscat_HOLIDAY_DATA_0_29 	: ARRAY [0..29] OF oscat_HOLIDAY_DATA;
END_TYPE

FUNCTION_BLOCK SETUP_HOLIDAY_FR_Block

	VAR_IN_OUT
		HD :	oscat_HOLIDAY_DATA_0_29;
	END_VAR

	VAR
		init :	BOOL;
	END_VAR

	IF init THEN RETURN; END_IF;

	init := TRUE;

	HD[00].NAME := 'Nouve an';
	HD[00].DAY  := SINT#01;
	HD[00].MONTH := SINT#01;
	HD[00].USE := SINT#01;

	HD[01].NAME := 'St Valentin';
	HD[01].DAY  := SINT#14;
	HD[01].MONTH := SINT#02;
	HD[01].USE := SINT#00;

	HD[02].NAME := 'Vendredi Saint (alsace)';
	HD[02].DAY  := SINT#-2;
	HD[02].MONTH := SINT#00;
	HD[02].USE := SINT#00;

	HD[03].NAME := 'Dimanche de pques';
	HD[03].DAY  := SINT#00;
	HD[03].MONTH := SINT#00;
	HD[03].USE := SINT#01;

	HD[04].NAME := 'Lundi de pques';
	HD[04].DAY  := SINT#01;
	HD[04].MONTH := SINT#00;
	HD[04].USE := SINT#01;

	HD[05].NAME := 'Jeudi de Ascension';
	HD[05].DAY  := SINT#39;
	HD[05].MONTH := SINT#00;
	HD[05].USE := SINT#01;

	HD[06].NAME := 'dimanche de Pentecte';
	HD[06].DAY  := SINT#49;
	HD[06].MONTH := SINT#00;
	HD[06].USE := SINT#01;

	HD[07].NAME := 'jeudi de la Trinit';
	HD[07].DAY  := SINT#60;
	HD[07].MONTH := SINT#00;
	HD[07].USE := SINT#00;

	HD[08].NAME := 'Fte du travail';
	HD[08].DAY  := SINT#01;
	HD[08].MONTH := SINT#05;
	HD[08].USE := SINT#01;

	HD[09].NAME := 'Victoire 1945 ';
	HD[09].DAY  := SINT#08;
	HD[09].MONTH := SINT#05;
	HD[09].USE := SINT#01;

	HD[10].NAME := 'Prise de La bastille';
	HD[10].DAY  := SINT#14;
	HD[10].MONTH := SINT#07;
	HD[10].USE := SINT#01;

	HD[11].NAME := '15 Aot 1944';
	HD[11].DAY  := SINT#15;
	HD[11].MONTH := SINT#08;
	HD[11].USE := SINT#01;

	HD[12].NAME := 'Halloween';
	HD[12].DAY  := SINT#31;
	HD[12].MONTH := SINT#10;
	HD[12].USE := SINT#00;

	HD[13].NAME := 'Armistice 1918';
	HD[13].DAY  := SINT#11;
	HD[13].MONTH := SINT#11;
	HD[13].USE := SINT#01;

	HD[14].NAME := 'Nol';
	HD[14].DAY  := SINT#25;
	HD[14].MONTH := SINT#12;
	HD[14].USE := SINT#01;

	HD[15].NAME := 'Saint tienne (alsace)';
	HD[15].DAY  := SINT#26;
	HD[15].MONTH := SINT#12;
	HD[15].USE := SINT#00;

	HD[16].NAME := 'Fte de la musique';
	HD[16].DAY  := SINT#21;
	HD[16].MONTH := SINT#06;
	HD[16].USE := SINT#00;
END_FUNCTION_BLOCK

PROGRAM program0
  VAR
    LocalVar0 : oscat_HOLIDAY_DATA_0_29;
	func_block : SETUP_HOLIDAY_FR_Block;
  END_VAR
	func_block.HD  := LocalVar0;
	func_block();
	LocalVar0 := func_block.HD;
END_PROGRAM

CONFIGURATION Config0
  RESOURCE Res0 ON PLC
    TASK task0(INTERVAL := T#20ms,PRIORITY := 0);
    PROGRAM instance0 WITH task0 : program0;
  END_RESOURCE
END_CONFIGURATION

(* ---- SETUP_LANGUAGE.ST ---- *)
TYPE oscat_LANGUAGE:
	STRUCT
		DEFAULT 	: INT;
		LMAX    	: INT;
	END_STRUCT;
END_TYPE

FUNCTION_BLOCK SETUP_LANGUAGE_Block

	VAR_IN_OUT
		LANGUAGE :	oscat_LANGUAGE;
	END_VAR

	VAR
		init :	BOOL;
	END_VAR

	IF init THEN RETURN; END_IF;
	init := TRUE;

	LANGUAGE.DEFAULT  := 1; (* 1=english, 2=german 3=french *)
	LANGUAGE.LMAX := 3;

END_FUNCTION_BLOCK

PROGRAM program0

	VAR
		LANGUAGE :	oscat_LANGUAGE;
		func_block : SETUP_LANGUAGE_Block;
	END_VAR
		func_block.LANGUAGE  := LANGUAGE;
		func_block();
		LANGUAGE := func_block.LANGUAGE;

END_PROGRAM

CONFIGURATION Config0

	RESOURCE Res0 ON PLC
		TASK task0(INTERVAL := T#20ms,PRIORITY := 0);
		PROGRAM instance0 WITH task0 : program0;
	END_RESOURCE

END_CONFIGURATION

(* ---- SETUP_LOCATION.ST ---- *)
TYPE
	oscat_LOCATION_ELEMENTS	: ARRAY [1..5] OF INT;
END_TYPE

TYPE oscat_LOCATION:
  STRUCT
    DEFAULT 	: INT;
	LMAX    	: INT;
	LANGUAGE	: oscat_LOCATION_ELEMENTS;
  END_STRUCT;
END_TYPE

FUNCTION_BLOCK SETUP_LOCATION_Block
	VAR_IN_OUT
		LOCATION :	oscat_LOCATION;
	END_VAR

	VAR
		init :	BOOL;
	END_VAR

	IF init THEN RETURN; END_IF;
	init := TRUE;

	LOCATION.DEFAULT  := 1;
	LOCATION.LMAX := 5;

	LOCATION.LANGUAGE[1] := 2;
	LOCATION.LANGUAGE[2] := 2;
	LOCATION.LANGUAGE[3] := 3;
	LOCATION.LANGUAGE[4] := 2;
	LOCATION.LANGUAGE[5] := 2;

END_FUNCTION_BLOCK

PROGRAM program0
	VAR
		LOCATION :	oscat_LOCATION;
		func_block : SETUP_LOCATION_Block;
  	END_VAR
	func_block.LOCATION  :=LOCATION;
	func_block();
	LOCATION := func_block.LOCATION;
END_PROGRAM

CONFIGURATION Config0
	RESOURCE Res0 ON PLC
		TASK task0(INTERVAL := T#20ms,PRIORITY := 0);
		PROGRAM instance0 WITH task0 : program0;
	END_RESOURCE
END_CONFIGURATION

(* ---- SETUP_MONTHS.ST ---- *)
TYPE
  oscat_ELEMENT_MONTHS 	: ARRAY [1..12] OF STRING;
  oscat_MONTHS			: ARRAY [1..3]  OF oscat_ELEMENT_MONTHS := [0, 0, 0];
END_TYPE

FUNCTION_BLOCK SETUP_MONTHS

	VAR_IN_OUT
		MONTHS :	oscat_MONTHS;
	END_VAR

	VAR
		init :	BOOL;
	END_VAR

	IF init THEN RETURN; END_IF;
	init := TRUE;

	(* ---- english --- *)
	MONTHS[1][01] := 'January';
	MONTHS[1][02] := 'February';
	MONTHS[1][03] := 'March';
	MONTHS[1][04] := 'April';
	MONTHS[1][05] := 'May';
	MONTHS[1][06] := 'June';
	MONTHS[1][07] := 'July';
	MONTHS[1][08] := 'August';
	MONTHS[1][09] := 'September';
	MONTHS[1][10] := 'October';
	MONTHS[1][11] := 'November';
	MONTHS[1][12] := 'December';

	(* ---- german --- *)
	MONTHS[2][01] := 'Januar';
	MONTHS[2][02] := 'Februar';
	MONTHS[2][03] := 'March';
	MONTHS[2][04] := 'April';
	MONTHS[2][05] := 'Mai';
	MONTHS[2][06] := 'Juni';
	MONTHS[2][07] := 'Juli';
	MONTHS[2][08] := 'August';
	MONTHS[2][09] := 'September';
	MONTHS[2][10] := 'Oktober';
	MONTHS[2][11] := 'November';
	MONTHS[2][12] := 'Dezember';

	(* ---- french --- *)
	MONTHS[3][01] := 'Janvier';
	MONTHS[3][02] := 'Fvrier';
	MONTHS[3][03] := 'mars';
	MONTHS[3][04] := 'Avril';
	MONTHS[3][05] := 'Mai';
	MONTHS[3][06] := 'Juin';
	MONTHS[3][07] := 'Juillet';
	MONTHS[3][08] := 'Aot';
	MONTHS[3][09] := 'Septembre';
	MONTHS[3][10] := 'Octobre';
	MONTHS[3][11] := 'Novembre';
	MONTHS[3][12] := 'Decembre';
END_FUNCTION_BLOCK

PROGRAM program0
  VAR
    LocalVar0 : oscat_MONTHS;
	func_block : SETUP_MONTHS;
  END_VAR
	func_block.MONTHS  := LocalVar0;
	func_block();
	LocalVar0 := func_block.MONTHS;
END_PROGRAM

CONFIGURATION Config0
  RESOURCE Res0 ON PLC
    TASK task0(INTERVAL := T#20ms,PRIORITY := 0);
    PROGRAM instance0 WITH task0 : program0;
  END_RESOURCE
END_CONFIGURATION

(* ---- SETUP_MONTHS3.ST ---- *)
TYPE
  oscat_ELEMENT_MONTHS3	: ARRAY [1..12] OF STRING;
  oscat_MONTHS3			: ARRAY [1..3]  OF oscat_ELEMENT_MONTHS3 := [0,0,0];
END_TYPE

FUNCTION_BLOCK SETUP_MONTHS3

	VAR_IN_OUT
		MONTHS3 :	oscat_MONTHS3;
	END_VAR

	VAR
		init :	BOOL;
	END_VAR

	IF init THEN RETURN; END_IF;
	init := TRUE;

	(* ---- english --- *)
	MONTHS3[1][01] := 'Jan';
	MONTHS3[1][02] := 'Feb';
	MONTHS3[1][03] := 'Mar';
	MONTHS3[1][04] := 'Apr';
	MONTHS3[1][05] := 'May';
	MONTHS3[1][06] := 'Jun';
	MONTHS3[1][07] := 'Jul';
	MONTHS3[1][08] := 'Aug';
	MONTHS3[1][09] := 'Sep';
	MONTHS3[1][10] := 'Oct';
	MONTHS3[1][11] := 'Nov';
	MONTHS3[1][12] := 'Dec';

	(* ---- german --- *)
	MONTHS3[2][01] := 'Jan';
	MONTHS3[2][02] := 'Feb';
	MONTHS3[2][03] := 'Mrz';
	MONTHS3[2][04] := 'Apr';
	MONTHs3[2][05] := 'Mai';
	MONTHS3[2][06] := 'Jun';
	MONTHS3[2][07] := 'Jul';
	MONTHS3[2][08] := 'Aug';
	MONTHS3[2][09] := 'Sep';
	MONTHS3[2][10] := 'Okt';
	MONTHS3[2][11] := 'Nov';
	MONTHS3[2][12] := 'Dez';

	(* ---- french --- *)
	MONTHS3[3][01] := 'Jan';
	MONTHS3[3][02] := 'Fev';
	MONTHS3[3][03] := 'Mar';
	MONTHS3[3][04] := 'Avr';
	MONTHs3[3][05] := 'Mai';
	MONTHS3[3][06] := 'Jun';
	MONTHS3[3][07] := 'Jul';
	MONTHS3[3][08] := 'Aou';
	MONTHS3[3][09] := 'Sep';
	MONTHS3[3][10] := 'Oct';
	MONTHS3[3][11] := 'Nov';
	MONTHS3[3][12] := 'Dec';
	(*@KEY@: END_WORKSHEET *)
	END_FUNCTION_BLOCK

PROGRAM program0
  VAR
    LocalVar0 : oscat_MONTHS3;
	func_block : SETUP_MONTHS3;
  END_VAR
	func_block.MONTHS3  := LocalVar0;
	func_block();
	LocalVar0 := func_block.MONTHS3;
END_PROGRAM

CONFIGURATION Config0
  RESOURCE Res0 ON PLC
    TASK task0(INTERVAL := T#20ms,PRIORITY := 0);
    PROGRAM instance0 WITH task0 : program0;
  END_RESOURCE
END_CONFIGURATION

(* ---- SETUP_WEEKDAYS.ST ---- *)
TYPE
  oscat_ELEMENT_WEEKDAYS	: ARRAY [1..7] OF STRING;
  oscat_WEEKDAYS			: ARRAY [1..3]  OF oscat_ELEMENT_WEEKDAYS := [0, 0, 0];
END_TYPE

FUNCTION_BLOCK SETUP_WEEKDAYS

	VAR_IN_OUT
		WEEKDAYS :	oscat_WEEKDAYS;
	END_VAR

	VAR
		init :	BOOL;
	END_VAR

	IF init THEN RETURN; END_IF;
	init := TRUE;

	WEEKDAYS[1][01] := 'Monday';
	WEEKDAYS[1][02] := 'Tuesday';
	WEEKDAYS[1][03] := 'Wednesday';
	WEEKDAYS[1][04] := 'Thursday';
	WEEKDAYS[1][05] := 'Friday';
	WEEKDAYS[1][06] := 'Saturday';
	WEEKDAYS[1][07] := 'Sunday';

	WEEKDAYS[2][01] := 'Montag';
	WEEKDAYS[2][02] := 'Dienstag';
	WEEKDAYS[2][03] := 'Mittwoch';
	WEEKDAYS[2][04] := 'Donnerstag';
	WEEKDAYS[2][05] := 'Freitag';
	WEEKDAYS[2][06] := 'Samstag';
	WEEKDAYS[2][07] := 'Sonntag';

	WEEKDAYS[3][01] := 'Lundi';
	WEEKDAYS[3][02] := 'Mardi';
	WEEKDAYS[3][03] := 'Mercredi';
	WEEKDAYS[3][04] := 'Jeudi';
	WEEKDAYS[3][05] := 'Vendredi';
	WEEKDAYS[3][06] := 'Samedi';
	WEEKDAYS[3][07] := 'Dimanche';
END_FUNCTION_BLOCK

PROGRAM program0
  VAR
    WEEKDAYS :	oscat_WEEKDAYS;
	func_block : SETUP_WEEKDAYS;
  END_VAR
	func_block.WEEKDAYS  := WEEKDAYS;
	func_block();
	WEEKDAYS := func_block.WEEKDAYS;

END_PROGRAM

CONFIGURATION Config0
  RESOURCE Res0 ON PLC
    TASK task0(INTERVAL := T#20ms,PRIORITY := 0);
    PROGRAM instance0 WITH task0 : program0;
  END_RESOURCE
END_CONFIGURATION

(* ---- SETUP_WEEKDAYS2.ST ---- *)
TYPE
  oscat_ELEMENT_WEEKDAYS2	: ARRAY [1..7] OF STRING;
  oscat_WEEKDAYS2			: ARRAY [1..3]  OF oscat_ELEMENT_WEEKDAYS2 := [0, 0, 0];
END_TYPE

FUNCTION_BLOCK SETUP_WEEKDAYS2_Block

	VAR_IN_OUT
		WEEKDAYS2 :	oscat_WEEKDAYS2;
	END_VAR

	VAR
		init :	BOOL;
	END_VAR

	IF init THEN RETURN; END_IF;
	init := TRUE;

	WEEKDAYS2[1][01] := 'Mo';
	WEEKDAYS2[1][02] := 'Tu';
	WEEKDAYS2[1][03] := 'We';
	WEEKDAYS2[1][04] := 'Th';
	WEEKDAYS2[1][05] := 'Fr';
	WEEKDAYS2[1][06] := 'Sa';
	WEEKDAYS2[1][07] := 'Su';

	WEEKDAYS2[2][01] := 'Mo';
	WEEKDAYS2[2][02] := 'Di';
	WEEKDAYS2[2][03] := 'Mi';
	WEEKDAYS2[2][04] := 'Do';
	WEEKDAYS2[2][05] := 'Fr';
	WEEKDAYS2[2][06] := 'Sa';
	WEEKDAYS2[2][07] := 'So';

	WEEKDAYS2[3][01] := 'Lu';
	WEEKDAYS2[3][02] := 'Ma';
	WEEKDAYS2[3][03] := 'Me';
	WEEKDAYS2[3][04] := 'Je';
	WEEKDAYS2[3][05] := 'Ve';
	WEEKDAYS2[3][06] := 'Sa';
	WEEKDAYS2[3][07] := 'Di';
END_FUNCTION_BLOCK

PROGRAM program0

	VAR
		WEEKDAYS2 :	oscat_WEEKDAYS2;
		func_block : SETUP_WEEKDAYS2_Block;
	END_VAR
		func_block.WEEKDAYS2 :=WEEKDAYS2;
		func_block();
		WEEKDAYS2 := func_block.WEEKDAYS2;

END_PROGRAM

CONFIGURATION Config0

	RESOURCE Res0 ON PLC
		TASK task0(INTERVAL := T#20ms,PRIORITY := 0);
		PROGRAM instance0 WITH task0 : program0;
	END_RESOURCE

END_CONFIGURATION

(* ---- SH.ST ---- *)
FUNCTION_BLOCK SH_Block

	VAR_INPUT
		IN :	REAL;
		CLK :	BOOL;
	END_VAR

	VAR_OUTPUT
		OUT :	REAL;
		TRIG :	BOOL;
	END_VAR

	VAR
		edge :	BOOL;
	END_VAR

	IF clk AND NOT edge THEN
		out := in;
		trig := TRUE;
	ELSE
		trig := FALSE;
	END_IF;
	edge := clk;

END_FUNCTION_BLOCK

PROGRAM program0

	VAR
		IN :	REAL;
		CLK :	BOOL;
		OUT :	REAL;
		TRIG :	BOOL;
		func_block : SH_Block;
	END_VAR
		func_block.IN  :=IN;
		func_block.CLK  :=CLK;
		func_block();
		OUT := func_block.OUT;
		TRIG := func_block.TRIG;

END_PROGRAM

CONFIGURATION Config0
	RESOURCE Res0 ON PLC
		TASK task0(INTERVAL := T#20ms,PRIORITY := 0);
		PROGRAM instance0 WITH task0 : program0;
	END_RESOURCE
END_CONFIGURATION

(* ---- SH_1.ST ---- *)
FUNCTION UDINT_TO_TIME2:TIME

	VAR_INPUT
		IN :	UDINT;
	END_VAR

	UDINT_TO_TIME2 := DINT_TO_TIME(UDINT_TO_DINT(IN));

END_FUNCTION

FUNCTION_BLOCK T_PLC_MS_block
	VAR_OUTPUT
		T_PLC_MS :	UDINT;
	END_VAR

	VAR_EXTERNAL
		PLC_TICKS_PER_SEC :	INT;
		PLC_SYS_TICK_CNT :	DINT;
	END_VAR

	VAR
		debug :	BOOL;(*Debug-Mode ON / OFF*)
		N :	INT;(*Debug-Faktor*)
		Offset :	UDINT;(*Debug-Offset*)
		temp :	DWORD := DWORD#1;(*Debug-Offset*)
		mode :	BOOL;(*modus*)
		faktor :	UDINT;(*Systemtakt-Faktor*)
		init :	BOOL;
		v_plc_ticks_per_sec :	UDINT;
		base :	UDINT := UDINT#1000;
	END_VAR

	IF init = FALSE THEN
		v_plc_ticks_per_sec := INT_TO_UDINT(PLC_TICKS_PER_SEC);
		IF v_plc_ticks_per_sec = UDINT#1024 THEN
			faktor := UDINT#1;
			mode := FALSE;
		ELSIF v_plc_ticks_per_sec > UDINT#0 THEN
			IF v_plc_ticks_per_sec <= base THEN
				faktor := base / v_plc_ticks_per_sec;
				mode := FALSE;
			ELSE
				faktor := v_plc_ticks_per_sec / base;
				mode := TRUE;
			END_IF;
		ELSE
			faktor := UDINT#1;
		END_IF;
		init := TRUE;
	END_IF;

	IF mode THEN
		T_PLC_MS := DINT_TO_UDINT(PLC_SYS_TICK_CNT) / faktor;
	ELSE
		T_PLC_MS := DINT_TO_UDINT(PLC_SYS_TICK_CNT) * faktor;
	END_IF;

	IF debug THEN
		T_PLC_MS := (DWORD_TO_UDINT(SHL(UDINT_TO_DWORD(T_PLC_MS),N) OR SHL(temp,N)) - UDINT#1) + Offset;
	END_IF;

END_FUNCTION_BLOCK

FUNCTION_BLOCK SH_1_Block

	VAR_INPUT
		IN :	REAL;
		PT :	TIME;
	END_VAR

	VAR_OUTPUT
		OUT :	REAL;
		TRIG :	BOOL;
	END_VAR

	VAR
		last :	TIME;
		tx :	TIME;
		T_PLC_MS :	T_PLC_MS_block;
	END_VAR

	T_PLC_MS();
	tx:= UDINT_TO_TIME(T_PLC_MS.T_PLC_MS);

	IF tx - last >= PT THEN
		last := tx;
		out := in;
		trig := TRUE;
	ELSE
		trig := FALSE;
	END_IF;

END_FUNCTION_BLOCK

PROGRAM program0

	VAR
		IN :	REAL;
		PT :	TIME;
		OUT :	REAL;
		TRIG :	BOOL;
		func_block : SH_1_Block;
	END_VAR
		func_block.IN  :=IN;
		func_block.PT  :=PT;
		func_block();
		OUT := func_block.OUT;
		TRIG := func_block.TRIG;

END_PROGRAM

CONFIGURATION Config0

	VAR_GLOBAL
		PLC_TICKS_PER_SEC :	INT;
		PLC_SYS_TICK_CNT :	DINT;
	END_VAR
	RESOURCE Res0 ON PLC
		TASK task0(INTERVAL := T#20ms,PRIORITY := 0);
		PROGRAM instance0 WITH task0 : program0;
	END_RESOURCE

END_CONFIGURATION

(* ---- SH_T.ST ---- *)
FUNCTION_BLOCK SH_T_Block

	VAR_INPUT
		IN :	REAL;
		E :	BOOL;
	END_VAR

	VAR_OUTPUT
		OUT :	REAL;
	END_VAR

	IF E THEN out := in; END_IF;

END_FUNCTION_BLOCK

PROGRAM program0

	VAR
		IN :	REAL;
		E :	BOOL;
		OUT :	REAL;
		func_block : SH_T_Block;
	END_VAR
	func_block.IN  :=IN;
	func_block.E  :=E;
	func_block();
	OUT := func_block.OUT;

END_PROGRAM

CONFIGURATION Config0

	RESOURCE Res0 ON PLC
		TASK task0(INTERVAL := T#20ms,PRIORITY := 0);
		PROGRAM instance0 WITH task0 : program0;
	END_RESOURCE

END_CONFIGURATION

(* ---- SHA1_STREAM.ST ---- *)
TYPE
  oscat_aB0_19	: ARRAY [0..19]	OF BYTE;
  oscat_aB0_63	: ARRAY [0..63]	OF BYTE;
  oscat_aDW0_4	: ARRAY [0..4] 	OF DWORD;
  oscat_sDW0_79	: ARRAY [0..79] OF DWORD;

END_TYPE

FUNCTION DWORD_OF_BYTE:DWORD
	VAR_INPUT
		B3 :	BYTE;
		B2 :	BYTE;
		B1 :	BYTE;
		B0 :	BYTE;
	END_VAR

	DWORD_OF_BYTE := SHL(SHL(SHL(BYTE_TO_DWORD(B3),8) OR BYTE_TO_DWORD(B2),8) OR BYTE_TO_DWORD(B1),8) OR BYTE_TO_DWORD(B0);

END_FUNCTION

FUNCTION_BLOCK SHA1_STREAM_Block

	VAR_IN_OUT
		MODE :	INT;
		BUF :	oscat_aB0_63;
		SHA1 :	oscat_aB0_19;
		SIZE :	UDINT;
	END_VAR

	VAR_OUTPUT
		POS :	UDINT;
	END_VAR

	VAR
		hash :	oscat_aDW0_4;
		end :	UDINT;
		block :	UDINT;
		pad_1 :	BOOL;
		w :	oscat_sDW0_79;
		n :	INT;
		n1 :	INT;
		n2 :	INT;
		n3 :	INT;
		n4 :	INT;
		a :	DWORD;
		b :	DWORD;
		c :	DWORD;
		d :	DWORD;
		e :	DWORD;
		f :	DWORD;
		k :	DWORD;
		x :	DWORD;
	END_VAR

	CASE MODE OF

	1:
		hash[0] := DWORD#16#67452301;
		hash[1] := DWORD#16#EFCDAB89;
		hash[2] := DWORD#16#98BADCFE;
		hash[3] := DWORD#16#10325476;
		hash[4] := DWORD#16#C3D2E1F0;

		FOR n := 16 TO 79 DO
			w[n] := DWORD#0;
		END_FOR;

		block := DWORD_TO_UDINT(SHR(UDINT_TO_DWORD(SIZE),6)) + BOOL_TO_UDINT((UDINT_TO_BYTE(SIZE) AND BYTE#16#3F) > BYTE#55);

		pad_1 := FALSE;
		POS := UDINT#0;
		End := SIZE;
		SIZE := MIN(UDINT#64,End);
		MODE := 2;

	2:	FOR n := UDINT_TO_INT(SIZE) TO 63 DO
			BUF[n] := BYTE#0;
		END_FOR;

		IF SIZE < UDINT#64 AND NOT pad_1 THEN
			BUF[SIZE] := BYTE#2#1000_0000;
			pad_1 := TRUE;
		END_IF;

		POS := POS + SIZE;
		SIZE := MIN(UDINT#64,End - POS);

		n := 0;
		FOR n4 := 0 TO 15 DO
			n1 := n + 1;
			n2 := n + 2;
			n3 := n + 3;
			w[n4] := DWORD_OF_BYTE(BUF[n],BUF[n1],BUF[n2],BUF[n3]);
			n := n + 4;
		END_FOR;

		IF block = UDINT#0 THEN
			w[15] := SHL(UDINT_TO_DWORD(End),3);
			MODE := 3;
		ELSE
			block := block - UDINT#1;
		END_IF;

		FOR n := 16 TO 79 DO
			n1 := n - 3;
			n2 := n - 8;
			n3 := n - 14;
			n4 := n - 16;
			w[n] := ROL(w[n1] XOR w[n2] XOR w[n3] XOR w[n4],1);
		END_FOR;

		a := hash[0];
		b := hash[1];
		c := hash[2];
		d := hash[3];
		e := hash[4];

		FOR n := 0 TO 79 DO
			IF n <= 19 THEN
				f := (b AND c) OR (NOT(b) AND d);
				k := DWORD#16#5A827999;
			ELSIF n <= 39 THEN
				f := b XOR c XOR d;
				k := DWORD#16#6ED9EBA1;
			ELSIF n <= 59 THEN
				f := (b AND c) OR (b AND d) OR (c AND d);
				k := DWORD#16#8F1BBCDC;
			ELSE
				f := b XOR c XOR d;
				k := DWORD#16#CA62C1D6;
			END_IF;

			x := UDINT_TO_DWORD(DWORD_TO_UDINT(ROL(a,5)) + DWORD_TO_UDINT(f) + DWORD_TO_UDINT(e) + DWORD_TO_UDINT(k) + DWORD_TO_UDINT(w[n]));
			e := d;
			d := c;
			c := ROL(b,30);
			b := a;
			a := x;
		END_FOR;

		hash[0] := UDINT_TO_DWORD(DWORD_TO_UDINT(hash[0]) + DWORD_TO_UDINT(a));
		hash[1] := UDINT_TO_DWORD(DWORD_TO_UDINT(hash[1]) + DWORD_TO_UDINT(b));
		hash[2] := UDINT_TO_DWORD(DWORD_TO_UDINT(hash[2]) + DWORD_TO_UDINT(c));
		hash[3] := UDINT_TO_DWORD(DWORD_TO_UDINT(hash[3]) + DWORD_TO_UDINT(d));
		hash[4] := UDINT_TO_DWORD(DWORD_TO_UDINT(hash[4]) + DWORD_TO_UDINT(e));

	END_CASE;

	IF MODE = 3 THEN
		n2 := 0;
		FOR n := 0 TO 4 DO
			FOR n1 := 0 TO 3 DO
				hash[n] := ROL(hash[n],8);
				SHA1[n2] := DWORD_TO_BYTE(hash[n]);
				n2 := n2 + 1;
			END_FOR;
		END_FOR;
	END_IF;

END_FUNCTION_BLOCK

PROGRAM program0
	VAR
		MODE :	INT;
		BUF :	oscat_aB0_63;
		SHA1 :	oscat_aB0_19;
		SIZE :	UDINT;
		POS :	UDINT;

		func_block : SHA1_STREAM_Block;
	END_VAR
	func_block.MODE := MODE;
	func_block.BUF := BUF;
	func_block.SHA1 := SHA1;
	func_block.SIZE := SIZE;

	func_block();
  	MODE  := func_block.MODE;
	BUF  := func_block.BUF;
	SHA1  := func_block.SHA1;
	SIZE  := func_block.SIZE;
	POS  := func_block.POS;
END_PROGRAM

CONFIGURATION Config0
	RESOURCE Res0 ON PLC
		TASK task0(INTERVAL := T#20ms,PRIORITY := 0);
		PROGRAM instance0 WITH task0 : program0;
	END_RESOURCE
END_CONFIGURATION

(* ---- SHR_4E.ST ---- *)
FUNCTION_BLOCK SHR_4E_Block

	VAR_INPUT
		SET :	BOOL;
		D0 :	BOOL;
		CLK :	BOOL;
		RST :	BOOL;
	END_VAR

	VAR_OUTPUT
		Q0 :	BOOL;
		Q1 :	BOOL;
		Q2 :	BOOL;
		Q3 :	BOOL;
	END_VAR

	VAR
		trig :	R_TRIG;
	END_VAR

	trig(clk := clk);

	IF set OR rst THEN
		Q0 := NOT RST;
		Q1 := Q0;
		Q2 := Q0;
		Q3 := Q0;
	ELSIF trig.Q THEN
		Q3 := Q2;
		Q2 := Q1;
		Q1 := Q0;
		Q0 := D0;
	END_IF;

END_FUNCTION_BLOCK

PROGRAM program0

	VAR
		SET :	BOOL;
		D0 :	BOOL;
		CLK :	BOOL;
		RST :	BOOL;
		Q0 :	BOOL;
		Q1 :	BOOL;
		Q2 :	BOOL;
		Q3 :	BOOL;
		func_block : SHR_4E_Block;
	END_VAR
	func_block.SET  :=SET;
	func_block.D0  :=D0;
	func_block.CLK  :=CLK;
	func_block.RST  :=RST;
	func_block();
	Q0 := func_block.Q0;
	Q1 := func_block.Q1;
	Q2 := func_block.Q2;
	Q3 := func_block.Q3;

END_PROGRAM

CONFIGURATION Config0
	RESOURCE Res0 ON PLC
		TASK task0(INTERVAL := T#20ms,PRIORITY := 0);
		PROGRAM instance0 WITH task0 : program0;
	END_RESOURCE
END_CONFIGURATION

(* ---- SHR_4UDE.ST ---- *)
FUNCTION_BLOCK SHR_4UDE_Block

	VAR_INPUT
		SET :	BOOL;
		D0 :	BOOL;
		D3 :	BOOL;
		CLK :	BOOL;
		DN :	BOOL;
		RST :	BOOL;
	END_VAR

	VAR_OUTPUT
		Q0 :	BOOL;
		Q1 :	BOOL;
		Q2 :	BOOL;
		Q3 :	BOOL;
	END_VAR

	VAR
		trig :	R_TRIG;
	END_VAR

	trig(clk := clk);

	IF set OR rst THEN
		Q0 := NOT RST;
		Q1 := Q0;
		Q2 := Q0;
		Q3 := Q0;
	ELSIF trig.Q THEN
		IF dn THEN
			Q0 := Q1;
			Q1 := Q2;
			Q2 := Q3;
			Q3 := D3;
		ELSE
			Q3 := Q2;
			Q2 := Q1;
			Q1 := Q0;
			Q0 := D0;
		END_IF;
	END_IF;

END_FUNCTION_BLOCK

PROGRAM program0

	VAR
		SET :	BOOL;
		D0 :	BOOL;
		D3 :	BOOL;
		CLK :	BOOL;
		DN :	BOOL;
		RST :	BOOL;
		Q0 :	BOOL;
		Q1 :	BOOL;
		Q2 :	BOOL;
		Q3 :	BOOL;
		func_block : SHR_4UDE_Block;
	END_VAR
	func_block.SET  :=SET;
	func_block.D0  :=D0;
	func_block.D3  :=D3;
	func_block.CLK  :=CLK;
	func_block.DN  :=DN;
	func_block.RST  :=RST;
	func_block();
	Q0 := func_block.Q0;
	Q1 := func_block.Q1;
	Q2 := func_block.Q2;
	Q3 := func_block.Q3;

END_PROGRAM

CONFIGURATION Config0
	RESOURCE Res0 ON PLC
		TASK task0(INTERVAL := T#20ms,PRIORITY := 0);
		PROGRAM instance0 WITH task0 : program0;
	END_RESOURCE
END_CONFIGURATION

(* ---- SHR_8PLE.ST ---- *)
FUNCTION BIT_OF_DWORD : BOOL
  VAR_INPUT
    IN : DWORD;
    N : INT;
  END_VAR

  BIT_OF_DWORD := (SHR(in,N) AND 16#00000001) > 0;
END_FUNCTION

FUNCTION BIT_LOAD_B:BYTE
	VAR_INPUT
		IN :	BYTE;
		VAL :	BOOL;
		POS :	INT;
	END_VAR

	IF VAL THEN
		BIT_LOAD_B := in OR SHL(BYTE#1,pos);
	ELSE
		BIT_LOAD_B := in AND (NOT SHL(BYTE#1,pos));
	END_IF;
END_FUNCTION

FUNCTION_BLOCK SHR_8PLE_Block

	VAR_INPUT
		DIN :	BOOL;
		DLOAD :	BYTE;
		CLK :	BOOL;
		UP :	BOOL := TRUE;
		LOAD :	BOOL;
		RST :	BOOL;
	END_VAR

	VAR_OUTPUT
		DOUT :	BOOL;
	END_VAR

	VAR
		edge :	BOOL := TRUE;
		register :	BYTE;
	END_VAR

	IF CLK AND edge AND NOT rst THEN
		edge := FALSE;
		IF UP THEN
			register := SHL(register,1);
			register := BIT_LOAD_B(register,Din,0);
			Dout     := BIT_OF_DWORD(BYTE_TO_DWORD(register),7);
		ELSE
			register := SHR(register,1);
			register := BIT_LOAD_B(register,Din,7);
			Dout     := BIT_OF_DWORD(BYTE_TO_DWORD(register),0);
		END_IF;
		IF load THEN
			register := Dload;
			IF up THEN
				Dout := BIT_OF_DWORD(BYTE_TO_DWORD(register),7);
			ELSE
				Dout := BIT_OF_DWORD(BYTE_TO_DWORD(register),0);
			END_IF;
		END_IF;
	END_IF;
	IF NOT clk THEN edge := TRUE; END_IF;
	IF rst THEN
		register := BYTE#0;
		Dout := FALSE;
	END_IF;

END_FUNCTION_BLOCK

PROGRAM program0
  	VAR
		DIN :	BOOL;
		DLOAD :	BYTE;
		CLK :	BOOL;
		UP :	BOOL := TRUE;
		LOAD :	BOOL;
		RST :	BOOL;
		DOUT :	BOOL;
		func_block : SHR_8PLE_Block;
	END_VAR
	func_block.DIN  :=DIN;
	func_block.DLOAD  :=DLOAD;
	func_block.CLK  :=CLK;
	func_block.UP  :=UP;
	func_block.LOAD  :=LOAD;
	func_block.RST  :=RST;
	func_block();
	DOUT := func_block.DOUT;

END_PROGRAM

CONFIGURATION Config0
	RESOURCE Res0 ON PLC
		TASK task0(INTERVAL := T#20ms,PRIORITY := 0);
		PROGRAM instance0 WITH task0 : program0;
	END_RESOURCE
END_CONFIGURATION

(* ---- SHR_8UDE.ST ---- *)
FUNCTION_BLOCK SHR_8UDE_Block

	VAR_INPUT
		SET :	BOOL;
		D0 :	BOOL;
		D7 :	BOOL;
		CLK :	BOOL;
		DN :	BOOL;
		RST :	BOOL;
	END_VAR

	VAR_OUTPUT
		Q0 :	BOOL;
		Q1 :	BOOL;
		Q2 :	BOOL;
		Q3 :	BOOL;
		Q4 :	BOOL;
		Q5 :	BOOL;
		Q6 :	BOOL;
		Q7 :	BOOL;
	END_VAR

	VAR
		trig :	R_TRIG;
	END_VAR

	trig(clk := clk);

	IF set OR rst THEN
		Q0 := NOT RST;
		Q1 := Q0;
		Q2 := Q0;
		Q3 := Q0;
		Q4 := Q0;
		Q5 := Q0;
		Q6 := Q0;
		Q7 := Q0;
	ELSIF trig.Q THEN
		IF dn THEN
			Q0 := Q1;
			Q1 := Q2;
			Q2 := Q3;
			Q3 := Q4;
			Q4 := Q5;
			Q5 := Q6;
			Q6 := Q7;
			Q7 := D7;
		ELSE
			Q7 := Q6;
			Q6 := Q5;
			Q5 := Q4;
			Q4 := Q3;
			Q3 := Q2;
			Q2 := Q1;
			Q1 := Q0;
			Q0 := D0;
		END_IF;
	END_IF;

END_FUNCTION_BLOCK

PROGRAM program0
	VAR
		SET :	BOOL;
		D0 :	BOOL;
		D7 :	BOOL;
		CLK :	BOOL;
		DN :	BOOL;
		RST :	BOOL;
		Q0 :	BOOL;
		Q1 :	BOOL;
		Q2 :	BOOL;
		Q3 :	BOOL;
		Q4 :	BOOL;
		Q5 :	BOOL;
		Q6 :	BOOL;
		Q7 :	BOOL;
		func_block : SHR_8UDE_Block;
  	END_VAR
	func_block.SET  :=SET;
	func_block.D0  :=D0;
	func_block.D7  :=D7;
	func_block.CLK  :=CLK;
	func_block.DN  :=DN;
	func_block.RST  :=RST;
	func_block();
	Q0  := func_block.Q0;
	Q1  := func_block.Q1;
	Q2  := func_block.Q2;
	Q3  := func_block.Q3;
	Q4  := func_block.Q4;
	Q5  := func_block.Q5;
	Q6  := func_block.Q6;
	Q7  := func_block.Q7;
END_PROGRAM

CONFIGURATION Config0
	RESOURCE Res0 ON PLC
		TASK task0(INTERVAL := T#20ms,PRIORITY := 0);
		PROGRAM instance0 WITH task0 : program0;
	END_RESOURCE
END_CONFIGURATION

(* ---- SIGNAL.ST ---- *)
FUNCTION _BYTE_TO_INT:INT
	VAR_INPUT
		IN :	BYTE;
	END_VAR

	_BYTE_TO_INT := USINT_TO_INT(BYTE_TO_USINT(IN));
END_FUNCTION

FUNCTION TIME_TO_UDINT2:UDINT
	VAR_INPUT
		X :	TIME;
	END_VAR

	TIME_TO_UDINT2 := DINT_TO_UDINT(TIME_TO_DINT(X));
END_FUNCTION

FUNCTION UDINT_TO_TIME2:TIME

	VAR_INPUT
		IN :	UDINT;
	END_VAR

	UDINT_TO_TIME2 := DINT_TO_TIME(UDINT_TO_DINT(IN));

END_FUNCTION

FUNCTION_BLOCK T_PLC_MS_block
	VAR_OUTPUT
		T_PLC_MS :	UDINT;
	END_VAR

	VAR_EXTERNAL
		PLC_TICKS_PER_SEC :	INT;
		PLC_SYS_TICK_CNT :	DINT;
	END_VAR

	VAR
		debug :	BOOL;(*Debug-Mode ON / OFF*)
		N :	INT;(*Debug-Faktor*)
		Offset :	UDINT;(*Debug-Offset*)
		temp :	DWORD := DWORD#1;(*Debug-Offset*)
		mode :	BOOL;(*modus*)
		faktor :	UDINT;(*Systemtakt-Faktor*)
		init :	BOOL;
		v_plc_ticks_per_sec :	UDINT;
		base :	UDINT := UDINT#1000;
	END_VAR

	IF init = FALSE THEN
		v_plc_ticks_per_sec := INT_TO_UDINT(PLC_TICKS_PER_SEC);
		IF v_plc_ticks_per_sec = UDINT#1024 THEN
			faktor := UDINT#1;
			mode := FALSE;
		ELSIF v_plc_ticks_per_sec > UDINT#0 THEN
			IF v_plc_ticks_per_sec <= base THEN
				faktor := base / v_plc_ticks_per_sec;
				mode := FALSE;
			ELSE
				faktor := v_plc_ticks_per_sec / base;
				mode := TRUE;
			END_IF;
		ELSE
			faktor := UDINT#1;
		END_IF;
		init := TRUE;
	END_IF;

	IF mode THEN
		T_PLC_MS := DINT_TO_UDINT(PLC_SYS_TICK_CNT) / faktor;
	ELSE
		T_PLC_MS := DINT_TO_UDINT(PLC_SYS_TICK_CNT) * faktor;
	END_IF;

	IF debug THEN
		T_PLC_MS := (DWORD_TO_UDINT(SHL(UDINT_TO_DWORD(T_PLC_MS),N) OR SHL(temp,N)) - UDINT#1) + Offset;
	END_IF;

END_FUNCTION_BLOCK

FUNCTION_BLOCK SIGNAL_Block

	VAR_INPUT
		IN :	BOOL;
		SIG :	BYTE;
		TS :	TIME;
	END_VAR

	VAR_OUTPUT
		Q :	BOOL;
	END_VAR

	VAR
		tx :	DWORD;
		_step :	BYTE;
		T_PLC_MS :	T_PLC_MS_Block;
	END_VAR

	IF in THEN
		T_PLC_MS();
		tx:= UDINT_TO_DWORD(T_PLC_MS.T_PLC_MS);

		IF ts > t#0s THEN
			_step := DWORD_TO_BYTE(UDINT_TO_DWORD(DWORD_TO_UDINT(tx) / TIME_TO_UDINT2(ts)) AND DWORD#16#0000_0007);
		ELSE
			_step := DWORD_TO_BYTE(SHR(tx,7) AND DWORD#16#0000_0007);
		END_IF;
		_step := SHL(BYTE#1,_BYTE_TO_INT(_step));
		Q := (_step AND sig) > BYTE#0;
	ELSE
		Q := FALSE;
	END_IF;

END_FUNCTION_BLOCK

PROGRAM program0
  VAR
	IN :	BOOL;
	SIG :	BYTE;
	TS :	TIME;
	Q :	BOOL;
	func_block : SIGNAL_Block;
  END_VAR
	func_block.IN  :=IN;
	func_block.SIG  :=SIG;
	func_block.TS  :=TS;
	func_block();
	Q := func_block.Q;

END_PROGRAM

CONFIGURATION Config0

	VAR_GLOBAL
		PLC_TICKS_PER_SEC :	INT;
		PLC_SYS_TICK_CNT :	DINT;
	END_VAR

  	RESOURCE Res0 ON PLC
    	TASK task0(INTERVAL := T#20ms,PRIORITY := 0);
    	PROGRAM instance0 WITH task0 : program0;
  	END_RESOURCE

END_CONFIGURATION

(* ---- SIGNAL_4.ST ---- *)
FUNCTION _BYTE_TO_INT:INT
	VAR_INPUT
		IN :	BYTE;
	END_VAR

	_BYTE_TO_INT := USINT_TO_INT(BYTE_TO_USINT(IN));
END_FUNCTION

FUNCTION TIME_TO_UDINT2:UDINT
	VAR_INPUT
		X :	TIME;
	END_VAR

	TIME_TO_UDINT2 := DINT_TO_UDINT(TIME_TO_DINT(X));
END_FUNCTION

FUNCTION UDINT_TO_TIME2:TIME

	VAR_INPUT
		IN :	UDINT;
	END_VAR

	UDINT_TO_TIME2 := DINT_TO_TIME(UDINT_TO_DINT(IN));

END_FUNCTION

FUNCTION_BLOCK T_PLC_MS_block
	VAR_OUTPUT
		T_PLC_MS :	UDINT;
	END_VAR

	VAR_EXTERNAL
		PLC_TICKS_PER_SEC :	INT;
		PLC_SYS_TICK_CNT :	DINT;
	END_VAR

	VAR
		debug :	BOOL;(*Debug-Mode ON / OFF*)
		N :	INT;(*Debug-Faktor*)
		Offset :	UDINT;(*Debug-Offset*)
		temp :	DWORD := DWORD#1;(*Debug-Offset*)
		mode :	BOOL;(*modus*)
		faktor :	UDINT;(*Systemtakt-Faktor*)
		init :	BOOL;
		v_plc_ticks_per_sec :	UDINT;
		base :	UDINT := UDINT#1000;
	END_VAR

	IF init = FALSE THEN
		v_plc_ticks_per_sec := INT_TO_UDINT(PLC_TICKS_PER_SEC);
		IF v_plc_ticks_per_sec = UDINT#1024 THEN
			faktor := UDINT#1;
			mode := FALSE;
		ELSIF v_plc_ticks_per_sec > UDINT#0 THEN
			IF v_plc_ticks_per_sec <= base THEN
				faktor := base / v_plc_ticks_per_sec;
				mode := FALSE;
			ELSE
				faktor := v_plc_ticks_per_sec / base;
				mode := TRUE;
			END_IF;
		ELSE
			faktor := UDINT#1;
		END_IF;
		init := TRUE;
	END_IF;

	IF mode THEN
		T_PLC_MS := DINT_TO_UDINT(PLC_SYS_TICK_CNT) / faktor;
	ELSE
		T_PLC_MS := DINT_TO_UDINT(PLC_SYS_TICK_CNT) * faktor;
	END_IF;

	IF debug THEN
		T_PLC_MS := (DWORD_TO_UDINT(SHL(UDINT_TO_DWORD(T_PLC_MS),N) OR SHL(temp,N)) - UDINT#1) + Offset;
	END_IF;

END_FUNCTION_BLOCK

FUNCTION_BLOCK SIGNAL_Block

	VAR_INPUT
		IN :	BOOL;
		SIG :	BYTE;
		TS :	TIME;
	END_VAR

	VAR_OUTPUT
		Q :	BOOL;
	END_VAR

	VAR
		tx :	DWORD;
		_step :	BYTE;
		T_PLC_MS :	T_PLC_MS_Block;
	END_VAR

	IF in THEN
		T_PLC_MS();
		tx:= UDINT_TO_DWORD(T_PLC_MS.T_PLC_MS);

		IF ts > t#0s THEN
			_step := DWORD_TO_BYTE(UDINT_TO_DWORD(DWORD_TO_UDINT(tx) / TIME_TO_UDINT2(ts)) AND DWORD#16#0000_0007);
		ELSE
			_step := DWORD_TO_BYTE(SHR(tx,7) AND DWORD#16#0000_0007);
		END_IF;
		_step := SHL(BYTE#1,_BYTE_TO_INT(_step));
		Q := (_step AND sig) > BYTE#0;
	ELSE
		Q := FALSE;
	END_IF;

END_FUNCTION_BLOCK

FUNCTION_BLOCK SIGNAL_4_Block

	VAR_INPUT
		IN1 :	BOOL;
		IN2 :	BOOL;
		IN3 :	BOOL;
		IN4 :	BOOL;
		TS :	TIME;
		S1 :	BYTE := 2#1111_1111;
		S2 :	BYTE := 2#1111_0000;
		S3 :	BYTE := 2#1010_1010;
		S4 :	BYTE := 2#1010_0000;
	END_VAR

	VAR_OUTPUT
		Q :	BOOL;
	END_VAR

	VAR
		sig :	SIGNAL_Block;
	END_VAR

	IF in1 THEN
		sig(in := TRUE, sig := s1, TS := TS);
	ELSIF in2 THEN
		sig(in := TRUE, sig := s2, TS := TS);
	ELSIF in3 THEN
		sig(in := TRUE, sig := s3, TS := TS);
	ELSIF in4 THEN
		sig(in := TRUE, sig := s4, TS := TS);
	ELSE
		sig(in := FALSE);
	END_IF;

	Q := sig.Q;

END_FUNCTION_BLOCK

PROGRAM program0

	VAR
		IN1 :	BOOL;
		IN2 :	BOOL;
		IN3 :	BOOL;
		IN4 :	BOOL;
		TS :	TIME;
		S1 :	BYTE := 2#1111_1111;
		S2 :	BYTE := 2#1111_0000;
		S3 :	BYTE := 2#1010_1010;
		S4 :	BYTE := 2#1010_0000;
		Q :	BOOL;
		func_block : SIGNAL_4_Block;
	END_VAR

	func_block.IN1  :=IN1;
	func_block.IN2  :=IN2;
	func_block.IN3  :=IN3;
	func_block.IN4  :=IN4;
	func_block.TS  :=TS;
	func_block.S1  :=S1;
	func_block.S2  :=S2;
	func_block.S3  :=S3;
	func_block.S4  :=S4;
	func_block();
	Q := func_block.Q;

END_PROGRAM

CONFIGURATION Config0

	VAR_GLOBAL
		PLC_TICKS_PER_SEC :	INT;
		PLC_SYS_TICK_CNT :	DINT;
	END_VAR

  	RESOURCE Res0 ON PLC
    	TASK task0(INTERVAL := T#20ms,PRIORITY := 0);
    	PROGRAM instance0 WITH task0 : program0;
  	END_RESOURCE

END_CONFIGURATION

(* ---- SNTP_CLIENT.ST ---- *)
TYPE
  oscat_IP_FIFO128_DATA  : ARRAY [1..128] OF BYTE;
  oscat_Mailbox  : ARRAY [1..16] OF BYTE;

  oscat_IP_FIFO_DATA :
  STRUCT
    X       : oscat_IP_FIFO128_DATA; (* IP_ID FIFO Speicher          *)
    Y       : oscat_IP_FIFO128_DATA; (* IP_ID Z�hler                 *)
    ID      : BYTE;                  (* h�chste vergabene id         *)
    MAX_ID  : BYTE;                  (* maximal Anmeldungen pro ID   *)
      INIT    : BOOL;                  (* Initialisierung durchgef�hrt *)
    EMPTY   : BOOL;                  (* FIFO leer                    *)
    FULL    : BOOL;                  (* FIFO voll                    *)
    TOP     : INT;                   (* maximale anzahl in FIFO      *)
    NW      : INT;                   (* Schreibzeiger                *)
    NR      : INT;                   (* Lesezeiger                   *)
  END_STRUCT;

  oscat_IP_C:
  STRUCT
    C_MODE:			BYTE;          		(*W Mode: TCP/UCP AKTIV/PASSIV                               *)
    C_PORT:         WORD;          		(*W Portnummer                                               *)
    C_IP:           DWORD;         		(*W IP-Adresse gepackt wwxxyyzz = www.xxx.yyy.zzz            *)
    C_STATE:        BYTE;          		(*R Verbindungsstatus ON/OFF + Flanke ON/OFF                 *)
    C_ENABLE:       BOOL;          		(*W Freigabe f�r Connect                                     *)
    R_OBSERVE:      BOOL;          		(*W Empfang ueberwachen                                      *)
    TIME_RESET:     BOOL;          		(*W Alle Timer ruecksetzen                                   *)
    ERROR:          DWORD;         		(*R vvwwxxyy (vv = CON_ERROR, ww = SEN_ERROR, xx = REC_ERROR *)
    FIFO:           oscat_IP_FIFO_DATA; (*I IP FIFO Struktur                                         *)
    MAILBOX:		oscat_Mailbox;		(*I Mailbox: Datenbereich f�r Bausteindatenaustausch         *)
  END_STRUCT;
END_TYPE

TYPE

  oscat_NW_BUF_LONG  : ARRAY [0..4095] OF BYTE;

  oscat_NETWORK_BUFFER :
  STRUCT
    SIZE   : UINT;
    BUFFER : oscat_NW_BUF_LONG;
  END_STRUCT;

END_TYPE

FUNCTION _BYTE_TO_INT:INT
	VAR_INPUT
		IN :	BYTE;
	END_VAR

	_BYTE_TO_INT := USINT_TO_INT(BYTE_TO_USINT(IN));
END_FUNCTION

FUNCTION_BLOCK IP_FIFO_Block

  VAR_IN_OUT
    FIFO :	oscat_IP_FIFO_DATA;
    ID :	BYTE;
    STATE :	BYTE;
  END_VAR

  VAR
    tmp :	INT;
  END_VAR

  IF NOT FIFO.INIT THEN
    FIFO.INIT		:= TRUE;
    FIFO.NW		:= 1;
    FIFO.NR		:= 1;
    FIFO.EMPTY	:= TRUE;
    FIFO.FULL		:= FALSE;
    FIFO.TOP		:= 128;
    FIFO.MAX_ID	:= BYTE#1;
  END_IF;

  IF ID = BYTE#00 THEN
    IF FIFO.ID < INT_TO_BYTE(FIFO.TOP) THEN
      ID := USINT_TO_BYTE(BYTE_TO_USINT(FIFO.ID) + USINT#1);
      FIFO.ID := ID ;

    ELSIF STATE < BYTE#200 THEN
      STATE := BYTE#255;
    RETURN;
    END_IF;
  END_IF;

  IF STATE = BYTE#1 AND NOT FIFO.FULL THEN
    tmp := _BYTE_TO_INT(ID);
    IF FIFO.Y[tmp] < FIFO.MAX_ID THEN
      FIFO.Y[tmp] := USINT_TO_BYTE(BYTE_TO_USINT(FIFO.Y[tmp]) + USINT#1);
      tmp := FIFO.NW;
      FIFO.X[tmp] := ID;
      IF FIFO.NW = FIFO.TOP THEN FIFO.NW := 1; ELSE FIFO.NW := FIFO.NW + 1; END_IF;
      FIFO.FULL := FIFO.NW = FIFO.NR;
    FIFO.EMPTY := FALSE;
      STATE := BYTE#2;
    END_IF;
  END_IF;

  IF STATE = BYTE#2 AND NOT FIFO.EMPTY THEN
    tmp := FIFO.NR;
    IF ID = FIFO.X[tmp] THEN
      STATE := BYTE#3;
    END_IF;
  END_IF;

  IF STATE = BYTE#4 AND NOT FIFO.EMPTY THEN

    tmp := FIFO.NR;
    IF ID = FIFO.X[tmp] THEN
      tmp := _BYTE_TO_INT(ID);
      FIFO.Y[tmp] := USINT_TO_BYTE(BYTE_TO_USINT(FIFO.Y[tmp]) - USINT#1);

      IF FIFO.NR = FIFO.TOP THEN FIFO.NR := 1; ELSE FIFO.NR := FIFO.NR + 1; END_IF;
      FIFO.EMPTY := FIFO.NR = FIFO.NW;
    FIFO.FULL := FALSE;
    END_IF;
    STATE := BYTE#5;
  END_IF;

END_FUNCTION_BLOCK

FUNCTION_BLOCK T_PLC_MS_block

	VAR_OUTPUT
		T_PLC_MS :	UDINT;
	END_VAR

	VAR_EXTERNAL
		PLC_TICKS_PER_SEC :	INT;
		PLC_SYS_TICK_CNT :	DINT;
	END_VAR

	VAR
		debug :	BOOL;(*Debug-Mode ON / OFF*)
		N :	INT;(*Debug-Faktor*)
		Offset :	UDINT;(*Debug-Offset*)
		temp :	DWORD := DWORD#1;(*Debug-Offset*)
		mode :	BOOL;(*modus*)
		faktor :	UDINT;(*Systemtakt-Faktor*)
		init :	BOOL;
		v_plc_ticks_per_sec :	UDINT;
		base :	UDINT := UDINT#1000;
	END_VAR

	IF init = FALSE THEN
		v_plc_ticks_per_sec := INT_TO_UDINT(PLC_TICKS_PER_SEC);
		IF v_plc_ticks_per_sec = UDINT#1024 THEN
			faktor := UDINT#1;
			mode := FALSE;
		ELSIF v_plc_ticks_per_sec > UDINT#0 THEN
			IF v_plc_ticks_per_sec <= base THEN
				faktor := base / v_plc_ticks_per_sec;
				mode := FALSE;
			ELSE
				faktor := v_plc_ticks_per_sec / base;
				mode := TRUE;
			END_IF;
		ELSE
			faktor := UDINT#1;
		END_IF;
		init := TRUE;
	END_IF;

	IF mode THEN
		T_PLC_MS := DINT_TO_UDINT(PLC_SYS_TICK_CNT) / faktor;
	ELSE
		T_PLC_MS := DINT_TO_UDINT(PLC_SYS_TICK_CNT) * faktor;
	END_IF;

	IF debug THEN
		T_PLC_MS := (DWORD_TO_UDINT(SHL(UDINT_TO_DWORD(T_PLC_MS),N) OR SHL(temp,N)) - UDINT#1) + Offset;
	END_IF;

END_FUNCTION_BLOCK

FUNCTION DWORD_OF_BYTE:DWORD
	VAR_INPUT
		B3 :	BYTE;
		B2 :	BYTE;
		B1 :	BYTE;
		B0 :	BYTE;
	END_VAR

	DWORD_OF_BYTE := SHL(SHL(SHL(BYTE_TO_DWORD(B3),8) OR BYTE_TO_DWORD(B2),8) OR BYTE_TO_DWORD(B1),8) OR BYTE_TO_DWORD(B0);

END_FUNCTION

FUNCTION _WORD_TO_DINT:DINT
	VAR_INPUT
		IN :	WORD;
	END_VAR
	_WORD_TO_DINT := UINT_TO_DINT(WORD_TO_UINT(IN));
END_FUNCTION

FUNCTION WORD_OF_BYTE:WORD
	VAR_INPUT
		B1 :	BYTE;
		B0 :	BYTE;
	END_VAR
	WORD_OF_BYTE := SHL(BYTE_TO_WORD(B1),8) OR BYTE_TO_WORD(B0);
END_FUNCTION

FUNCTION _INT_TO_UDINT:UDINT
	VAR_INPUT
		IN :	INT;
	END_VAR

	_INT_TO_UDINT := DINT_TO_UDINT(INT_TO_DINT(IN));
END_FUNCTION

FUNCTION_BLOCK SNTP_CLIENT_Block

  VAR_IN_OUT
    IP_C :	oscat_IP_C;
    S_BUF :	oscat_NETWORK_BUFFER;
    R_BUF :	oscat_NETWORK_BUFFER;
  END_VAR

  VAR_INPUT
    IP4 :	DWORD;
    ACTIVATE :	BOOL;
  END_VAR

  VAR_OUTPUT
    ERROR :	DWORD;
    DONE_P :	BOOL;
    UDT :	UDINT;
    XMS :	INT;
  END_VAR

  VAR
    IP_STATE :	BYTE;
    IP_ID :	BYTE;
    IP_FIFO :	IP_FIFO_Block;
    i :	INT;
    last :	UDINT;
    state :	INT;
    T_PLC_MS :	T_PLC_MS_Block;
    tx :	UDINT;
    ACTIVATE_LAST :	BOOL;
    IP4_STORED :	DWORD;
  END_VAR

  T_PLC_MS();
  tx := T_PLC_MS.T_PLC_MS;

  CASE state OF
  00:
    DONE_P := FALSE;
    IF ACTIVATE AND NOT ACTIVATE_LAST THEN
      IP4_STORED := IP4;
      state := 10;
      ERROR := DWORD#0;
      IP_STATE := BYTE#1;
    END_IF;

  10:
    IF IP_STATE = BYTE#3 THEN

      S_BUF.BUFFER[00] := BYTE#16#1B;
      FOR i := 1 TO 47 DO
        S_BUF.BUFFER[i] := BYTE#16#00;
      END_FOR;

      last := tx;
      state := 30;

      IP_C.C_PORT     := WORD#123;
      IP_C.C_IP       := IP4_STORED;
      IP_C.C_MODE     := BYTE#1;
      IP_C.C_ENABLE   := TRUE;
      IP_C.TIME_RESET := TRUE;
      IP_C.R_OBSERVE  := TRUE;
      S_BUF.SIZE      := UINT#48;
      R_BUF.SIZE      := UINT#0;
    END_IF;

  30:
    IF IP_C.ERROR <> DWORD#00 THEN
      ERROR := IP_C.ERROR;
    S_BUF.SIZE := UINT#0;
    R_BUF.SIZE := UINT#0;
      state := 0;
    ELSIF S_BUF.SIZE = UINT#0 AND R_BUF.SIZE >= UINT#48 THEN
      UDT := DWORD_TO_UDINT(DWORD_OF_BYTE(R_BUF.BUFFER[40],R_BUF.BUFFER[41],R_BUF.BUFFER[42],R_BUF.BUFFER[43]))- UDINT#2208988800;

      XMS := DWORD_TO_INT(SHR(DINT_TO_DWORD(_WORD_TO_DINT(WORD_OF_BYTE(R_BUF.BUFFER[44],R_BUF.BUFFER[45])) * DINT#1000),16));
      XMS := XMS + DWORD_TO_INT(SHR(UDINT_TO_DWORD(tx - last),1));

      UDT := UDT + _INT_TO_UDINT(XMS / 1000);
      XMS := XMS MOD 1000;

      state := 0;
      DONE_P := TRUE;

    END_IF;

    IF state = 0 THEN
      IP_C.R_OBSERVE := FALSE;
      IP_STATE := BYTE#4;
    END_IF;

  END_CASE;

  ACTIVATE_LAST := ACTIVATE;

  IP_FIFO(FIFO:=IP_C.FIFO,STATE:=IP_STATE,ID:=IP_ID);
  IP_C.FIFO:=IP_FIFO.FIFO;
  IP_STATE := IP_FIFO.STATE;
  IP_ID:=IP_FIFO.ID;

END_FUNCTION_BLOCK

PROGRAM program0
	VAR
		IP_C :	oscat_IP_C;
    S_BUF :	oscat_NETWORK_BUFFER;
    R_BUF :	oscat_NETWORK_BUFFER;
    IP4 :	DWORD;
    ACTIVATE :	BOOL;
    ERROR :	DWORD;
    DONE_P :	BOOL;
    UDT :	UDINT;
    XMS :	INT;

		func_block : SNTP_CLIENT_Block;
	END_VAR
	func_block.IP_C := IP_C;
	func_block.S_BUF := S_BUF;
	func_block.R_BUF := R_BUF;
  func_block.IP4 := IP4;
	func_block.ACTIVATE := ACTIVATE;

	func_block();
  IP_C  := func_block.IP_C;
  S_BUF  := func_block.S_BUF;
  R_BUF  := func_block.R_BUF;
  ERROR  := func_block.ERROR;
  DONE_P  := func_block.DONE_P;
  UDT  := func_block.UDT;
  XMS  := func_block.XMS;
END_PROGRAM

CONFIGURATION Config0

	VAR_GLOBAL
		PLC_TICKS_PER_SEC :	INT;
		PLC_SYS_TICK_CNT :	DINT;
	END_VAR

  	RESOURCE Res0 ON PLC
    	TASK task0(INTERVAL := T#20ms,PRIORITY := 0);
    	PROGRAM instance0 WITH task0 : program0;
  	END_RESOURCE

END_CONFIGURATION

(* ---- SPEED.ST ---- *)
FUNCTION_BLOCK SPEED_Block

	VAR_INPUT
		MS :	REAL;
		KMH :	REAL;
		KN :	REAL;
		MH :	REAL;
	END_VAR

	VAR_OUTPUT
		YMS :	REAL;
		YKMH :	REAL;
		YKN :	REAL;
		YMH :	REAL;
	END_VAR

	Yms := ms +
			kmh * 0.27777777777778 +
			kn * 0.5144444 +
			mh * 0.44704;
	Ykmh := Yms * 3.6;
	Ykn := Yms * 1.94384466037535;
	Ymh := Yms * 2.23693629205440;

END_FUNCTION_BLOCK

PROGRAM program0

	VAR
		MS :	REAL;
		KMH :	REAL;
		KN :	REAL;
		MH :	REAL;
		YMS :	REAL;
		YKMH :	REAL;
		YKN :	REAL;
		YMH :	REAL;
		func_block : SPEED_Block;
	END_VAR
		func_block.MS  :=MS;
		func_block.KMH  :=KMH;
		func_block.KN  :=KN;
		func_block.MH  :=MH;
		func_block();
		YMS := func_block.YMS;
		YKMH := func_block.YKMH;
		YKN := func_block.YKN;
		YMH := func_block.YMH;

	END_PROGRAM

CONFIGURATION Config0

	RESOURCE Res0 ON PLC
		TASK task0(INTERVAL := T#20ms,PRIORITY := 0);
		PROGRAM instance0 WITH task0 : program0;
	END_RESOURCE

END_CONFIGURATION
